LIN {X 0,Y 351.942,Z 392.186,A -85,B 0,C 180,E1 14008.468,E2 14008.468} C_VEL
LIN {X 0,Y 334.172,Z 595.574,A -85,B 0,C 180,E1 14003.413,E2 14003.413} C_VEL
LIN {X 0,Y 330.821,Z 619.274,A -85,B 0,C 180,E1 14002.569,E2 14002.569} C_VEL
LIN {X 0,Y 326.72,Z 641.204,A -85,B 0,C 180,E1 14001.516,E2 14001.516} C_VEL
LIN {X 0,Y 321.807,Z 663.482,A -85,B 0,C 180,E1 14000.12,E2 14000.12} C_VEL
LIN {X 0,Y 316.522,Z 684.324,A -85,B 0,C 180,E1 13998.471,E2 13998.471} C_VEL
LIN {X 0,Y 310.9,Z 704.371,A -85,B 0,C 180,E1 13996.508,E2 13996.508} C_VEL
LIN {X 0,Y 304.922,Z 723.772,A -85,B 0,C 180,E1 13994.168,E2 13994.168} C_VEL
LIN {X 0,Y 299.118,Z 741.54,A -85,B 0,C 180,E1 13991.566,E2 13991.566} C_VEL
LIN {X 0,Y 293.223,Z 758.965,A -85,B 0,C 180,E1 13988.482,E2 13988.482} C_VEL
LIN {X 0,Y 288.236,Z 773.54,A -85,B 0,C 180,E1 13985.391,E2 13985.391} C_VEL
LIN {X 0,Y 283.487,Z 787.604,A -85,B 0,C 180,E1 13981.785,E2 13981.785} C_VEL
LIN {X 0,Y 279.718,Z 799.334,A -85,B 0,C 180,E1 13978.151,E2 13978.151} C_VEL
LIN {X 0,Y 276.584,Z 810.131,A -85,B 0,C 180,E1 13974.108,E2 13974.108} C_VEL
LIN {X 0,Y 274.424,Z 818.988,A -85,B 0,C 180,E1 13970.026,E2 13970.026} C_VEL
LIN {X 0,Y 273.126,Z 825.97,A -85,B 0,C 180,E1 13965.933,E2 13965.933} C_VEL
LIN {X 0,Y 272.509,Z 831.598,A -85,B 0,C 180,E1 13961.64,E2 13961.64} C_VEL
LIN {X 0,Y 272.417,Z 835.097,A -85,B 0,C 180,E1 13957.803,E2 13957.803} C_VEL
LIN {X 0,Y 272.52,Z 837.318,A -85,B 0,C 180,E1 13953.784,E2 13953.784} C_VEL
LIN {X 0,Y 272.599,Z 837.937,A -85,B 0,C 180,E1 13950.208,E2 13950.208} C_VEL
LIN {X 0,Y 272.53,Z 837.335,A -85,B 0,C 180,E1 13946.422,E2 13946.422} C_VEL
LIN {X 0,Y 272.421,Z 835.096,A -85,B 0,C 180,E1 13942.405,E2 13942.405} C_VEL
LIN {X 0,Y 272.503,Z 831.449,A -85,B 0,C 180,E1 13938.356,E2 13938.356} C_VEL
LIN {X 0,Y 273.106,Z 825.844,A -85,B 0,C 180,E1 13934.061,E2 13934.061} C_VEL
LIN {X 0,Y 274.571,Z 818.159,A -85,B 0,C 180,E1 13929.536,E2 13929.536} C_VEL
LIN {X 0,Y 276.978,Z 808.952,A -85,B 0,C 180,E1 13925.243,E2 13925.243} C_VEL
LIN {X 0,Y 280.51,Z 797.735,A -85,B 0,C 180,E1 13921.001,E2 13921.001} C_VEL
LIN {X 0,Y 285.267,Z 784.462,A -85,B 0,C 180,E1 13916.852,E2 13916.852} C_VEL
LIN {X 0,Y 290.991,Z 769.791,A -85,B 0,C 180,E1 13913.034,E2 13913.034} C_VEL
LIN {X 0,Y 298.348,Z 751.957,A -85,B 0,C 180,E1 13909.192,E2 13909.192} C_VEL
LIN {X 0,Y 307.129,Z 731.579,A -85,B 0,C 180,E1 13905.577,E2 13905.577} C_VEL
LIN {X 0,Y 316.878,Z 709.867,A -85,B 0,C 180,E1 13902.407,E2 13902.407} C_VEL
LIN {X 0,Y 327.837,Z 686.66,A -85,B 0,C 180,E1 13899.636,E2 13899.636} C_VEL
LIN {X 0,Y 339.629,Z 663.013,A -85,B 0,C 180,E1 13897.355,E2 13897.355} C_VEL
LIN {X 0,Y 346.995,Z 648.595,A -85,B 0,C 180,E1 13896.209,E2 13896.209} C_VEL
LIN {X 0,Y 335.989,Z 668.452,A -85,B 0,C 180,E1 13894.02,E2 13894.02} C_VEL
LIN {X 0,Y 324.563,Z 689.118,A -85,B 0,C 180,E1 13891.17,E2 13891.17} C_VEL
LIN {X 0,Y 315.027,Z 706.467,A -85,B 0,C 180,E1 13888.225,E2 13888.225} C_VEL
LIN {X 0,Y 305.764,Z 723.244,A -85,B 0,C 180,E1 13884.746,E2 13884.746} C_VEL
LIN {X 0,Y 298.466,Z 736.332,A -85,B 0,C 180,E1 13881.419,E2 13881.419} C_VEL
LIN {X 0,Y 291.857,Z 748.263,A -85,B 0,C 180,E1 13877.755,E2 13877.755} C_VEL
LIN {X 0,Y 286.081,Z 758.861,A -85,B 0,C 180,E1 13873.751,E2 13873.751} C_VEL
LIN {X 0,Y 281.081,Z 768.361,A -85,B 0,C 180,E1 13869.214,E2 13869.214} C_VEL
LIN {X 0,Y 277.403,Z 775.806,A -85,B 0,C 180,E1 13864.551,E2 13864.551} C_VEL
LIN {X 0,Y 275.095,Z 780.905,A -85,B 0,C 180,E1 13860.211,E2 13860.211} C_VEL
LIN {X 0,Y 273.648,Z 784.687,A -85,B 0,C 180,E1 13855.602,E2 13855.602} C_VEL
LIN {X 0,Y 272.931,Z 786.813,A -85,B 0,C 180,E1 13851.152,E2 13851.152} C_VEL
LIN {X 0,Y 272.65,Z 787.32,A -85,B 0,C 180,E1 13847.077,E2 13847.077} C_VEL
LIN {X 0,Y 272.588,Z 786.619,A -85,B 0,C 180,E1 13842.939,E2 13842.939} C_VEL
LIN {X 0,Y 272.677,Z 784.598,A -85,B 0,C 180,E1 13838.943,E2 13838.943} C_VEL
LIN {X 0,Y 273.155,Z 780.795,A -85,B 0,C 180,E1 13834.414,E2 13834.414} C_VEL
LIN {X 0,Y 274.12,Z 775.808,A -85,B 0,C 180,E1 13830.243,E2 13830.243} C_VEL
LIN {X 0,Y 275.777,Z 769.08,A -85,B 0,C 180,E1 13826.063,E2 13826.063} C_VEL
LIN {X 0,Y 278.331,Z 760.51,A -85,B 0,C 180,E1 13821.843,E2 13821.843} C_VEL
LIN {X 0,Y 281.677,Z 750.53,A -85,B 0,C 180,E1 13817.87,E2 13817.87} C_VEL
LIN {X 0,Y 285.732,Z 739.008,A -85,B 0,C 180,E1 13814.138,E2 13814.138} C_VEL
LIN {X 0,Y 290.521,Z 725.684,A -85,B 0,C 180,E1 13810.578,E2 13810.578} C_VEL
LIN {X 0,Y 296.06,Z 710.191,A -85,B 0,C 180,E1 13807.159,E2 13807.159} C_VEL
LIN {X 0,Y 301.439,Z 694.762,A -85,B 0,C 180,E1 13804.325,E2 13804.325} C_VEL
LIN {X 0,Y 307.215,Z 677.128,A -85,B 0,C 180,E1 13801.637,E2 13801.637} C_VEL
LIN {X 0,Y 312.723,Z 658.939,A -85,B 0,C 180,E1 13799.343,E2 13799.343} C_VEL
LIN {X 0,Y 318.43,Z 638.248,A -85,B 0,C 180,E1 13797.194,E2 13797.194} C_VEL
LIN {X 0,Y 323.465,Z 617.601,A -85,B 0,C 180,E1 13795.448,E2 13795.448} C_VEL
LIN {X 0,Y 327.941,Z 596.27,A -85,B 0,C 180,E1 13793.992,E2 13793.992} C_VEL
LIN {X 0,Y 331.872,Z 573.214,A -85,B 0,C 180,E1 13792.774,E2 13792.774} C_VEL
LIN {X 0,Y 334.859,Z 550.767,A -85,B 0,C 180,E1 13791.893,E2 13791.893} C_VEL
LIN {X 0,Y 337.662,Z 520.747,A -85,B 0,C 180,E1 13791.075,E2 13791.075} C_VEL
LIN {X 0,Y 349.694,Z 379.97,A -85,B 0,C 180,E1 13787.623,E2 13787.623} C_VEL
LIN {X 0,Y 338.542,Z 362.97,A -85,B 0,C 180,E1 13784.541,E2 13784.541} C_VEL
LIN {X 0,Y 328.746,Z 348.783,A -85,B 0,C 180,E1 13781.553,E2 13781.553} C_VEL
LIN {X 0,Y 319.208,Z 335.537,A -85,B 0,C 180,E1 13778.335,E2 13778.335} C_VEL
LIN {X 0,Y 311.113,Z 324.801,A -85,B 0,C 180,E1 13775.303,E2 13775.303} C_VEL
LIN {X 0,Y 307.024,Z 319.574,A -85,B 0,C 180,E1 13773.69,E2 13773.69} C_VEL
LIN {X 0,Y 303.123,Z 314.492,A -85,B 0,C 180,E1 13772.013,E2 13772.013} C_VEL
LIN {X 0,Y 298.721,Z 308.948,A -85,B 0,C 180,E1 13770.055,E2 13770.055} C_VEL
LIN {X 0,Y 295.301,Z 304.475,A -85,B 0,C 180,E1 13768.401,E2 13768.401} C_VEL
LIN {X 0,Y 290.911,Z 299.407,A -85,B 0,C 180,E1 13766.208,E2 13766.208} C_VEL
LIN {X 0,Y 289.799,Z 297.619,A -85,B 0,C 180,E1 13765.583,E2 13765.583} C_VEL
LIN {X 0,Y 286.586,Z 294.45,A -85,B 0,C 180,E1 13763.855,E2 13763.855} C_VEL
LIN {X 0,Y 284.817,Z 291.431,A -85,B 0,C 180,E1 13762.742,E2 13762.742} C_VEL
LIN {X 0,Y 281.599,Z 288.767,A -85,B 0,C 180,E1 13760.911,E2 13760.911} C_VEL
LIN {X 0,Y 279.649,Z 285.071,A -85,B 0,C 180,E1 13759.472,E2 13759.472} C_VEL
LIN {X 0,Y 276.423,Z 282.89,A -85,B 0,C 180,E1 13757.468,E2 13757.468} C_VEL
LIN {X 0,Y 274.693,Z 279.757,A -85,B 0,C 180,E1 13756.048,E2 13756.048} C_VEL
LIN {X 0,Y 274.436,Z 278.542,A -85,B 0,C 180,E1 13755.658,E2 13755.658} C_VEL
LIN {X 0,Y 274.453,Z 278.534,A -85,B 0,C 180,E1 13750.862,E2 13750.862} C_VEL
LIN {X 0,Y 274.454,Z 278.532,A -85,B 0,C 180,E1 13746.15,E2 13746.15} C_VEL
LIN {X 0,Y 274.433,Z 278.536,A -85,B 0,C 180,E1 13741.4,E2 13741.4} C_VEL
LIN {X 0,Y 274.449,Z 278.537,A -85,B 0,C 180,E1 13736.628,E2 13736.628} C_VEL
LIN {X 0,Y 274.445,Z 278.542,A -85,B 0,C 180,E1 13731.893,E2 13731.893} C_VEL
LIN {X 0,Y 274.427,Z 278.549,A -85,B 0,C 180,E1 13727.077,E2 13727.077} C_VEL
LIN {X 0,Y 274.45,Z 278.55,A -85,B 0,C 180,E1 13722.31,E2 13722.31} C_VEL
LIN {X 0,Y 274.443,Z 278.549,A -85,B 0,C 180,E1 13717.734,E2 13717.734} C_VEL
LIN {X 0,Y 274.423,Z 278.554,A -85,B 0,C 180,E1 13712.876,E2 13712.876} C_VEL
LIN {X 0,Y 274.445,Z 278.55,A -85,B 0,C 180,E1 13708.163,E2 13708.163} C_VEL
LIN {X 0,Y 274.429,Z 278.552,A -85,B 0,C 180,E1 13703.351,E2 13703.351} C_VEL
LIN {X 0,Y 274.442,Z 278.55,A -85,B 0,C 180,E1 13699.818,E2 13699.818} C_VEL
LIN {X 0,Y 273.594,Z 278.663,A -85,B 0,C 180,E1 13698.323,E2 13698.323} C_VEL
LIN {X 0,Y 269.921,Z 279.115,A -85,B 0,C 180,E1 13695.846,E2 13695.846} C_VEL
LIN {X 0,Y 266.816,Z 279.496,A -85,B 0,C 180,E1 13693.407,E2 13693.407} C_VEL
LIN {X 0,Y 266.475,Z 279.543,A -85,B 0,C 180,E1 13692.444,E2 13692.444} C_VEL
LIN {X 0,Y 266.523,Z 279.674,A -85,B 0,C 180,E1 13687.704,E2 13687.704} C_VEL
LIN {X 0,Y 267.429,Z 282.454,A -85,B 0,C 180,E1 13686.545,E2 13686.545} C_VEL
LIN {X 0,Y 270.123,Z 285.3,A -85,B 0,C 180,E1 13684.243,E2 13684.243} C_VEL
LIN {X 0,Y 272.079,Z 286.502,A -85,B 0,C 180,E1 13682.788,E2 13682.788} C_VEL
LIN {X 0,Y 274,Z 290.15,A -85,B 0,C 180,E1 13681.121,E2 13681.121} C_VEL
LIN {X 0,Y 277.469,Z 293.008,A -85,B 0,C 180,E1 13678.758,E2 13678.758} C_VEL
LIN {X 0,Y 279.723,Z 296.759,A -85,B 0,C 180,E1 13677.129,E2 13677.129} C_VEL
LIN {X 0,Y 282.798,Z 299.497,A -85,B 0,C 180,E1 13675.282,E2 13675.282} C_VEL
LIN {X 0,Y 285.389,Z 303.379,A -85,B 0,C 180,E1 13673.661,E2 13673.661} C_VEL
LIN {X 0,Y 287.285,Z 305.462,A -85,B 0,C 180,E1 13672.599,E2 13672.599} C_VEL
LIN {X 0,Y 291.204,Z 310.688,A -85,B 0,C 180,E1 13670.412,E2 13670.412} C_VEL
LIN {X 0,Y 295.841,Z 316.996,A -85,B 0,C 180,E1 13668.051,E2 13668.051} C_VEL
LIN {X 0,Y 302.81,Z 326.638,A -85,B 0,C 180,E1 13664.779,E2 13664.779} C_VEL
LIN {X 0,Y 312.198,Z 340.01,A -85,B 0,C 180,E1 13660.834,E2 13660.834} C_VEL
LIN {X 0,Y 322.538,Z 355.803,A -85,B 0,C 180,E1 13656.958,E2 13656.958} C_VEL
LIN {X 0,Y 332.5,Z 371.552,A -85,B 0,C 180,E1 13653.62,E2 13653.62} C_VEL
LIN {X 0,Y 343.151,Z 389.583,A -85,B 0,C 180,E1 13650.378,E2 13650.378} C_VEL
LIN {X 0,Y 346.545,Z 395.753,A -85,B 0,C 180,E1 13649.4,E2 13649.4} C_VEL
LIN {X 0,Y 328.463,Z 594.891,A -85,B 0,C 180,E1 13644.391,E2 13644.391} C_VEL
LIN {X 0,Y 324.989,Z 618.714,A -85,B 0,C 180,E1 13643.533,E2 13643.533} C_VEL
LIN {X 0,Y 320.71,Z 640.907,A -85,B 0,C 180,E1 13642.457,E2 13642.457} C_VEL
LIN {X 0,Y 315.639,Z 663.183,A -85,B 0,C 180,E1 13641.045,E2 13641.045} C_VEL
LIN {X 0,Y 310.162,Z 684.106,A -85,B 0,C 180,E1 13639.367,E2 13639.367} C_VEL
LIN {X 0,Y 304.352,Z 704.148,A -85,B 0,C 180,E1 13637.379,E2 13637.379} C_VEL
LIN {X 0,Y 298.224,Z 723.376,A -85,B 0,C 180,E1 13635.022,E2 13635.022} C_VEL
LIN {X 0,Y 292.219,Z 741.11,A -85,B 0,C 180,E1 13632.378,E2 13632.378} C_VEL
LIN {X 0,Y 286.097,Z 758.503,A -85,B 0,C 180,E1 13629.236,E2 13629.236} C_VEL
LIN {X 0,Y 280.773,Z 773.445,A -85,B 0,C 180,E1 13625.982,E2 13625.982} C_VEL
LIN {X 0,Y 276.01,Z 787.001,A -85,B 0,C 180,E1 13622.418,E2 13622.418} C_VEL
LIN {X 0,Y 271.94,Z 799.128,A -85,B 0,C 180,E1 13618.551,E2 13618.551} C_VEL
LIN {X 0,Y 268.556,Z 810.359,A -85,B 0,C 180,E1 13614.173,E2 13614.173} C_VEL
LIN {X 0,Y 266.376,Z 819.075,A -85,B 0,C 180,E1 13609.97,E2 13609.97} C_VEL
LIN {X 0,Y 265.086,Z 825.898,A -85,B 0,C 180,E1 13605.755,E2 13605.755} C_VEL
LIN {X 0,Y 264.51,Z 831.309,A -85,B 0,C 180,E1 13601.334,E2 13601.334} C_VEL
LIN {X 0,Y 264.453,Z 834.685,A -85,B 0,C 180,E1 13597.383,E2 13597.383} C_VEL
LIN {X 0,Y 264.572,Z 836.606,A -85,B 0,C 180,E1 13593.464,E2 13593.464} C_VEL
LIN {X 0,Y 264.645,Z 837.141,A -85,B 0,C 180,E1 13589.998,E2 13589.998} C_VEL
LIN {X 0,Y 264.552,Z 836.49,A -85,B 0,C 180,E1 13586.097,E2 13586.097} C_VEL
LIN {X 0,Y 264.439,Z 834.34,A -85,B 0,C 180,E1 13582.164,E2 13582.164} C_VEL
LIN {X 0,Y 264.522,Z 830.928,A -85,B 0,C 180,E1 13578.22,E2 13578.22} C_VEL
LIN {X 0,Y 265.211,Z 825.167,A -85,B 0,C 180,E1 13573.573,E2 13573.573} C_VEL
LIN {X 0,Y 266.716,Z 817.962,A -85,B 0,C 180,E1 13569.135,E2 13569.135} C_VEL
LIN {X 0,Y 269.273,Z 808.87,A -85,B 0,C 180,E1 13564.72,E2 13564.72} C_VEL
LIN {X 0,Y 273.259,Z 797.259,A -85,B 0,C 180,E1 13560.136,E2 13560.136} C_VEL
LIN {X 0,Y 278.636,Z 783.539,A -85,B 0,C 180,E1 13555.708,E2 13555.708} C_VEL
LIN {X 0,Y 285.158,Z 768.226,A -85,B 0,C 180,E1 13551.637,E2 13551.637} C_VEL
LIN {X 0,Y 293.535,Z 749.713,A -85,B 0,C 180,E1 13547.587,E2 13547.587} C_VEL
LIN {X 0,Y 303.996,Z 727.824,A -85,B 0,C 180,E1 13543.688,E2 13543.688} C_VEL
LIN {X 0,Y 315.653,Z 704.899,A -85,B 0,C 180,E1 13540.375,E2 13540.375} C_VEL
LIN {X 0,Y 327.969,Z 682.1,A -85,B 0,C 180,E1 13537.708,E2 13537.708} C_VEL
LIN {X 0,Y 337.842,Z 664.742,A -85,B 0,C 180,E1 13536.037,E2 13536.037} C_VEL
LIN {X 0,Y 325.213,Z 684.979,A -85,B 0,C 180,E1 13533.392,E2 13533.392} C_VEL
LIN {X 0,Y 313.431,Z 704.056,A -85,B 0,C 180,E1 13530.269,E2 13530.269} C_VEL
LIN {X 0,Y 302.725,Z 721.589,A -85,B 0,C 180,E1 13526.694,E2 13526.694} C_VEL
LIN {X 0,Y 293.873,Z 736.129,A -85,B 0,C 180,E1 13523.036,E2 13523.036} C_VEL
LIN {X 0,Y 286.647,Z 748.093,A -85,B 0,C 180,E1 13519.354,E2 13519.354} C_VEL
LIN {X 0,Y 279.981,Z 759.214,A -85,B 0,C 180,E1 13515.114,E2 13515.114} C_VEL
LIN {X 0,Y 274.435,Z 768.713,A -85,B 0,C 180,E1 13510.499,E2 13510.499} C_VEL
LIN {X 0,Y 270.449,Z 775.926,A -85,B 0,C 180,E1 13505.944,E2 13505.944} C_VEL
LIN {X 0,Y 267.672,Z 781.44,A -85,B 0,C 180,E1 13501.287,E2 13501.287} C_VEL
LIN {X 0,Y 266.015,Z 785.203,A -85,B 0,C 180,E1 13496.771,E2 13496.771} C_VEL
LIN {X 0,Y 265.136,Z 787.339,A -85,B 0,C 180,E1 13492.419,E2 13492.419} C_VEL
LIN {X 0,Y 264.721,Z 788.143,A -85,B 0,C 180,E1 13487.792,E2 13487.792} C_VEL
LIN {X 0,Y 264.624,Z 787.62,A -85,B 0,C 180,E1 13483.767,E2 13483.767} C_VEL
LIN {X 0,Y 264.686,Z 785.665,A -85,B 0,C 180,E1 13479.436,E2 13479.436} C_VEL
LIN {X 0,Y 265.091,Z 782.273,A -85,B 0,C 180,E1 13475.015,E2 13475.015} C_VEL
LIN {X 0,Y 266.004,Z 777.39,A -85,B 0,C 180,E1 13470.7,E2 13470.7} C_VEL
LIN {X 0,Y 267.726,Z 770.585,A -85,B 0,C 180,E1 13466.193,E2 13466.193} C_VEL
LIN {X 0,Y 270.302,Z 762.203,A -85,B 0,C 180,E1 13461.853,E2 13461.853} C_VEL
LIN {X 0,Y 273.697,Z 752.363,A -85,B 0,C 180,E1 13457.769,E2 13457.769} C_VEL
LIN {X 0,Y 277.793,Z 741.088,A -85,B 0,C 180,E1 13453.963,E2 13453.963} C_VEL
LIN {X 0,Y 282.93,Z 727.351,A -85,B 0,C 180,E1 13450.142,E2 13450.142} C_VEL
LIN {X 0,Y 288.379,Z 712.726,A -85,B 0,C 180,E1 13446.789,E2 13446.789} C_VEL
LIN {X 0,Y 294.323,Z 696.294,A -85,B 0,C 180,E1 13443.671,E2 13443.671} C_VEL
LIN {X 0,Y 300.189,Z 678.978,A -85,B 0,C 180,E1 13440.97,E2 13440.97} C_VEL
LIN {X 0,Y 305.923,Z 660.788,A -85,B 0,C 180,E1 13438.611,E2 13438.611} C_VEL
LIN {X 0,Y 311.642,Z 640.918,A -85,B 0,C 180,E1 13436.483,E2 13436.483} C_VEL
LIN {X 0,Y 316.902,Z 620.387,A -85,B 0,C 180,E1 13434.687,E2 13434.687} C_VEL
LIN {X 0,Y 321.588,Z 598.842,A -85,B 0,C 180,E1 13433.181,E2 13433.181} C_VEL
LIN {X 0,Y 325.565,Z 576.701,A -85,B 0,C 180,E1 13431.964,E2 13431.964} C_VEL
LIN {X 0,Y 328.935,Z 553.047,A -85,B 0,C 180,E1 13430.989,E2 13430.989} C_VEL
LIN {X 0,Y 331.69,Z 525.923,A -85,B 0,C 180,E1 13430.213,E2 13430.213} C_VEL
LIN {X 0,Y 344.309,Z 383.812,A -85,B 0,C 180,E1 13426.688,E2 13426.688} C_VEL
LIN {X 0,Y 332.876,Z 366.29,A -85,B 0,C 180,E1 13423.4,E2 13423.4} C_VEL
LIN {X 0,Y 322.598,Z 351.536,A -85,B 0,C 180,E1 13420.132,E2 13420.132} C_VEL
LIN {X 0,Y 312.829,Z 337.953,A -85,B 0,C 180,E1 13416.66,E2 13416.66} C_VEL
LIN {X 0,Y 304.199,Z 326.687,A -85,B 0,C 180,E1 13413.252,E2 13413.252} C_VEL
LIN {X 0,Y 300.032,Z 321.302,A -85,B 0,C 180,E1 13411.442,E2 13411.442} C_VEL
LIN {X 0,Y 295.841,Z 315.95,A -85,B 0,C 180,E1 13409.527,E2 13409.527} C_VEL
LIN {X 0,Y 291.65,Z 310.532,A -85,B 0,C 180,E1 13407.448,E2 13407.448} C_VEL
LIN {X 0,Y 288.18,Z 306.433,A -85,B 0,C 180,E1 13405.674,E2 13405.674} C_VEL
LIN {X 0,Y 286.993,Z 304.767,A -85,B 0,C 180,E1 13405.005,E2 13405.005} C_VEL
LIN {X 0,Y 283.721,Z 301.163,A -85,B 0,C 180,E1 13403.176,E2 13403.176} C_VEL
LIN {X 0,Y 282.258,Z 298.807,A -85,B 0,C 180,E1 13402.266,E2 13402.266} C_VEL
LIN {X 0,Y 279.069,Z 295.873,A -85,B 0,C 180,E1 13400.36,E2 13400.36} C_VEL
LIN {X 0,Y 277.159,Z 292.56,A -85,B 0,C 180,E1 13398.979,E2 13398.979} C_VEL
LIN {X 0,Y 273.841,Z 289.901,A -85,B 0,C 180,E1 13396.811,E2 13396.811} C_VEL
LIN {X 0,Y 271.834,Z 286.096,A -85,B 0,C 180,E1 13395.082,E2 13395.082} C_VEL
LIN {X 0,Y 268.572,Z 283.959,A -85,B 0,C 180,E1 13392.675,E2 13392.675} C_VEL
LIN {X 0,Y 266.903,Z 281.204,A -85,B 0,C 180,E1 13391.038,E2 13391.038} C_VEL
LIN {X 0,Y 266.52,Z 279.52,A -85,B 0,C 180,E1 13390.498,E2 13390.498} C_VEL
LIN {X 0,Y 266.498,Z 279.523,A -85,B 0,C 180,E1 13385.731,E2 13385.731} C_VEL
LIN {X 0,Y 266.508,Z 279.527,A -85,B 0,C 180,E1 13380.812,E2 13380.812} C_VEL
LIN {X 0,Y 266.507,Z 279.533,A -85,B 0,C 180,E1 13376.002,E2 13376.002} C_VEL
LIN {X 0,Y 266.489,Z 279.542,A -85,B 0,C 180,E1 13371.205,E2 13371.205} C_VEL
LIN {X 0,Y 266.51,Z 279.544,A -85,B 0,C 180,E1 13366.349,E2 13366.349} C_VEL
LIN {X 0,Y 266.495,Z 279.547,A -85,B 0,C 180,E1 13361.607,E2 13361.607} C_VEL
LIN {X 0,Y 266.492,Z 279.542,A -85,B 0,C 180,E1 13356.596,E2 13356.596} C_VEL
LIN {X 0,Y 266.509,Z 279.537,A -85,B 0,C 180,E1 13351.933,E2 13351.933} C_VEL
LIN {X 0,Y 266.486,Z 279.536,A -85,B 0,C 180,E1 13347.23,E2 13347.23} C_VEL
LIN {X 0,Y 266.492,Z 279.531,A -85,B 0,C 180,E1 13342.265,E2 13342.265} C_VEL
LIN {X 0,Y 266.492,Z 279.528,A -85,B 0,C 180,E1 13337.463,E2 13337.463} C_VEL
LIN {X 0,Y 266.474,Z 279.543,A -85,B 0,C 180,E1 13332.566,E2 13332.566} C_VEL
LIN {X 0,Y 266.475,Z 279.543,A -85,B 0,C 180,E1 13332.444,E2 13332.444} C_VEL
LIN {X 0,Y 266.106,Z 280.303,A -85,B 0,C 180,E1 13331.338,E2 13331.338} C_VEL
LIN {X 0,Y 264.864,Z 283.505,A -85,B 0,C 180,E1 13329.703,E2 13329.703} C_VEL
LIN {X 0,Y 264.474,Z 287.92,A -85,B 0,C 180,E1 13327.957,E2 13327.957} C_VEL
LIN {X 0,Y 264.679,Z 288.591,A -85,B 0,C 180,E1 13327.663,E2 13327.663} C_VEL
LIN {X 0,Y 266.748,Z 291.851,A -85,B 0,C 180,E1 13325.59,E2 13325.59} C_VEL
LIN {X 0,Y 269.783,Z 294.028,A -85,B 0,C 180,E1 13323.237,E2 13323.237} C_VEL
LIN {X 0,Y 272.021,Z 297.888,A -85,B 0,C 180,E1 13321.333,E2 13321.333} C_VEL
LIN {X 0,Y 275.163,Z 300.601,A -85,B 0,C 180,E1 13319.164,E2 13319.164} C_VEL
LIN {X 0,Y 277.712,Z 304.517,A -85,B 0,C 180,E1 13317.315,E2 13317.315} C_VEL
LIN {X 0,Y 280.388,Z 306.967,A -85,B 0,C 180,E1 13315.703,E2 13315.703} C_VEL
LIN {X 0,Y 283.392,Z 311.177,A -85,B 0,C 180,E1 13313.82,E2 13313.82} C_VEL
LIN {X 0,Y 285.203,Z 313.416,A -85,B 0,C 180,E1 13312.787,E2 13312.787} C_VEL
LIN {X 0,Y 288.592,Z 317.897,A -85,B 0,C 180,E1 13310.883,E2 13310.883} C_VEL
LIN {X 0,Y 293.267,Z 324.376,A -85,B 0,C 180,E1 13308.443,E2 13308.443} C_VEL
LIN {X 0,Y 299.789,Z 333.498,A -85,B 0,C 180,E1 13305.314,E2 13305.314} C_VEL
LIN {X 0,Y 308.896,Z 346.614,A -85,B 0,C 180,E1 13301.405,E2 13301.405} C_VEL
LIN {X 0,Y 318.934,Z 362.103,A -85,B 0,C 180,E1 13297.56,E2 13297.56} C_VEL
LIN {X 0,Y 328.594,Z 377.505,A -85,B 0,C 180,E1 13294.253,E2 13294.253} C_VEL
LIN {X 0,Y 339.211,Z 395.689,A -85,B 0,C 180,E1 13290.945,E2 13290.945} C_VEL
LIN {X 0,Y 341.176,Z 399.501,A -85,B 0,C 180,E1 13290.351,E2 13290.351} C_VEL
LIN {X 0,Y 322.724,Z 594.496,A -85,B 0,C 180,E1 13285.377,E2 13285.377} C_VEL
LIN {X 0,Y 319.149,Z 618.283,A -85,B 0,C 180,E1 13284.511,E2 13284.511} C_VEL
LIN {X 0,Y 314.705,Z 640.646,A -85,B 0,C 180,E1 13283.415,E2 13283.415} C_VEL
LIN {X 0,Y 309.548,Z 662.612,A -85,B 0,C 180,E1 13282.008,E2 13282.008} C_VEL
LIN {X 0,Y 303.765,Z 684.004,A -85,B 0,C 180,E1 13280.269,E2 13280.269} C_VEL
LIN {X 0,Y 297.664,Z 704.298,A -85,B 0,C 180,E1 13278.216,E2 13278.216} C_VEL
LIN {X 0,Y 291.356,Z 723.49,A -85,B 0,C 180,E1 13275.823,E2 13275.823} C_VEL
LIN {X 0,Y 285.164,Z 741.146,A -85,B 0,C 180,E1 13273.132,E2 13273.132} C_VEL
LIN {X 0,Y 279.019,Z 757.975,A -85,B 0,C 180,E1 13270.03,E2 13270.03} C_VEL
LIN {X 0,Y 273.654,Z 772.52,A -85,B 0,C 180,E1 13266.81,E2 13266.81} C_VEL
LIN {X 0,Y 268.603,Z 786.3,A -85,B 0,C 180,E1 13263.115,E2 13263.115} C_VEL
LIN {X 0,Y 264.381,Z 798.3,A -85,B 0,C 180,E1 13259.197,E2 13259.197} C_VEL
LIN {X 0,Y 260.964,Z 809.063,A -85,B 0,C 180,E1 13254.924,E2 13254.924} C_VEL
LIN {X 0,Y 258.605,Z 817.905,A -85,B 0,C 180,E1 13250.597,E2 13250.597} C_VEL
LIN {X 0,Y 257.196,Z 824.874,A -85,B 0,C 180,E1 13246.209,E2 13246.209} C_VEL
LIN {X 0,Y 256.557,Z 830.34,A -85,B 0,C 180,E1 13241.69,E2 13241.69} C_VEL
LIN {X 0,Y 256.484,Z 833.764,A -85,B 0,C 180,E1 13237.614,E2 13237.614} C_VEL
LIN {X 0,Y 256.607,Z 835.774,A -85,B 0,C 180,E1 13233.572,E2 13233.572} C_VEL
LIN {X 0,Y 256.686,Z 836.331,A -85,B 0,C 180,E1 13229.998,E2 13229.998} C_VEL
LIN {X 0,Y 256.591,Z 835.761,A -85,B 0,C 180,E1 13226.2,E2 13226.2} C_VEL
LIN {X 0,Y 256.454,Z 833.617,A -85,B 0,C 180,E1 13221.929,E2 13221.929} C_VEL
LIN {X 0,Y 256.556,Z 830.211,A -85,B 0,C 180,E1 13217.849,E2 13217.849} C_VEL
LIN {X 0,Y 257.324,Z 824.493,A -85,B 0,C 180,E1 13213.055,E2 13213.055} C_VEL
LIN {X 0,Y 258.988,Z 817.376,A -85,B 0,C 180,E1 13208.482,E2 13208.482} C_VEL
LIN {X 0,Y 261.763,Z 808.355,A -85,B 0,C 180,E1 13203.941,E2 13203.941} C_VEL
LIN {X 0,Y 266.045,Z 796.958,A -85,B 0,C 180,E1 13199.26,E2 13199.26} C_VEL
LIN {X 0,Y 271.52,Z 784.19,A -85,B 0,C 180,E1 13194.936,E2 13194.936} C_VEL
LIN {X 0,Y 278.383,Z 769.264,A -85,B 0,C 180,E1 13190.79,E2 13190.79} C_VEL
LIN {X 0,Y 287.176,Z 751.446,A -85,B 0,C 180,E1 13186.692,E2 13186.692} C_VEL
LIN {X 0,Y 297.926,Z 730.952,A -85,B 0,C 180,E1 13182.834,E2 13182.834} C_VEL
LIN {X 0,Y 310.558,Z 708.587,A -85,B 0,C 180,E1 13179.402,E2 13179.402} C_VEL
LIN {X 0,Y 323.711,Z 686.923,A -85,B 0,C 180,E1 13176.722,E2 13176.722} C_VEL
LIN {X 0,Y 328.633,Z 679.199,A -85,B 0,C 180,E1 13175.863,E2 13175.863} C_VEL
LIN {X 0,Y 314.914,Z 698.765,A -85,B 0,C 180,E1 13172.885,E2 13172.885} C_VEL
LIN {X 0,Y 302.762,Z 716.583,A -85,B 0,C 180,E1 13169.479,E2 13169.479} C_VEL
LIN {X 0,Y 292.236,Z 732.229,A -85,B 0,C 180,E1 13165.757,E2 13165.757} C_VEL
LIN {X 0,Y 283.193,Z 745.764,A -85,B 0,C 180,E1 13161.762,E2 13161.762} C_VEL
LIN {X 0,Y 275.284,Z 757.737,A -85,B 0,C 180,E1 13157.33,E2 13157.33} C_VEL
LIN {X 0,Y 269.153,Z 767.239,A -85,B 0,C 180,E1 13152.881,E2 13152.881} C_VEL
LIN {X 0,Y 264.403,Z 774.959,A -85,B 0,C 180,E1 13148.265,E2 13148.265} C_VEL
LIN {X 0,Y 260.831,Z 781.171,A -85,B 0,C 180,E1 13143.299,E2 13143.299} C_VEL
LIN {X 0,Y 258.611,Z 785.354,A -85,B 0,C 180,E1 13138.452,E2 13138.452} C_VEL
LIN {X 0,Y 257.406,Z 787.89,A -85,B 0,C 180,E1 13133.759,E2 13133.759} C_VEL
LIN {X 0,Y 256.858,Z 788.991,A -85,B 0,C 180,E1 13129.234,E2 13129.234} C_VEL
LIN {X 0,Y 256.672,Z 788.625,A -85,B 0,C 180,E1 13124.874,E2 13124.874} C_VEL
LIN {X 0,Y 256.689,Z 787.009,A -85,B 0,C 180,E1 13120.432,E2 13120.432} C_VEL
LIN {X 0,Y 256.979,Z 784.029,A -85,B 0,C 180,E1 13116.116,E2 13116.116} C_VEL
LIN {X 0,Y 257.809,Z 779.365,A -85,B 0,C 180,E1 13111.513,E2 13111.513} C_VEL
LIN {X 0,Y 259.338,Z 773.318,A -85,B 0,C 180,E1 13107.074,E2 13107.074} C_VEL
LIN {X 0,Y 261.762,Z 765.344,A -85,B 0,C 180,E1 13102.608,E2 13102.608} C_VEL
LIN {X 0,Y 265.107,Z 755.766,A -85,B 0,C 180,E1 13098.313,E2 13098.313} C_VEL
LIN {X 0,Y 269.31,Z 744.602,A -85,B 0,C 180,E1 13094.236,E2 13094.236} C_VEL
LIN {X 0,Y 274.328,Z 731.727,A -85,B 0,C 180,E1 13090.387,E2 13090.387} C_VEL
LIN {X 0,Y 279.898,Z 717.262,A -85,B 0,C 180,E1 13086.859,E2 13086.859} C_VEL
LIN {X 0,Y 285.852,Z 701.374,A -85,B 0,C 180,E1 13083.652,E2 13083.652} C_VEL
LIN {X 0,Y 292.049,Z 684.074,A -85,B 0,C 180,E1 13080.767,E2 13080.767} C_VEL
LIN {X 0,Y 298.102,Z 665.944,A -85,B 0,C 180,E1 13078.262,E2 13078.262} C_VEL
LIN {X 0,Y 304.016,Z 646.359,A -85,B 0,C 180,E1 13076.044,E2 13076.044} C_VEL
LIN {X 0,Y 309.507,Z 625.976,A -85,B 0,C 180,E1 13074.163,E2 13074.163} C_VEL
LIN {X 0,Y 314.667,Z 603.891,A -85,B 0,C 180,E1 13072.521,E2 13072.521} C_VEL
LIN {X 0,Y 318.897,Z 582.26,A -85,B 0,C 180,E1 13071.248,E2 13071.248} C_VEL
LIN {X 0,Y 322.505,Z 559.319,A -85,B 0,C 180,E1 13070.214,E2 13070.214} C_VEL
LIN {X 0,Y 325.24,Z 535.374,A -85,B 0,C 180,E1 13069.455,E2 13069.455} C_VEL
LIN {X 0,Y 338.861,Z 387.588,A -85,B 0,C 180,E1 13065.731,E2 13065.731} C_VEL
LIN {X 0,Y 328.152,Z 371.194,A -85,B 0,C 180,E1 13062.54,E2 13062.54} C_VEL
LIN {X 0,Y 318.86,Z 357.651,A -85,B 0,C 180,E1 13059.477,E2 13059.477} C_VEL
LIN {X 0,Y 309.53,Z 344.557,A -85,B 0,C 180,E1 13056.074,E2 13056.074} C_VEL
LIN {X 0,Y 300.959,Z 333.282,A -85,B 0,C 180,E1 13052.62,E2 13052.62} C_VEL
LIN {X 0,Y 296.847,Z 327.999,A -85,B 0,C 180,E1 13050.83,E2 13050.83} C_VEL
LIN {X 0,Y 292.983,Z 322.945,A -85,B 0,C 180,E1 13048.994,E2 13048.994} C_VEL
LIN {X 0,Y 288.847,Z 317.623,A -85,B 0,C 180,E1 13046.926,E2 13046.926} C_VEL
LIN {X 0,Y 285.302,Z 313.162,A -85,B 0,C 180,E1 13045.026,E2 13045.026} C_VEL
LIN {X 0,Y 283.712,Z 311.406,A -85,B 0,C 180,E1 13044.136,E2 13044.136} C_VEL
LIN {X 0,Y 280.414,Z 307.115,A -85,B 0,C 180,E1 13042.215,E2 13042.215} C_VEL
LIN {X 0,Y 279.529,Z 306.031,A -85,B 0,C 180,E1 13041.673,E2 13041.673} C_VEL
LIN {X 0,Y 276.397,Z 302.752,A -85,B 0,C 180,E1 13039.698,E2 13039.698} C_VEL
LIN {X 0,Y 274.804,Z 300.066,A -85,B 0,C 180,E1 13038.565,E2 13038.565} C_VEL
LIN {X 0,Y 271.525,Z 297.2,A -85,B 0,C 180,E1 13036.322,E2 13036.322} C_VEL
LIN {X 0,Y 269.545,Z 293.678,A -85,B 0,C 180,E1 13034.661,E2 13034.661} C_VEL
LIN {X 0,Y 266.356,Z 291.339,A -85,B 0,C 180,E1 13032.188,E2 13032.188} C_VEL
LIN {X 0,Y 264.518,Z 288.257,A -85,B 0,C 180,E1 13030.402,E2 13030.402} C_VEL
LIN {X 0,Y 264.056,Z 287.139,A -85,B 0,C 180,E1 13029.882,E2 13029.882} C_VEL
LIN {X 0,Y 260.718,Z 285.035,A -85,B 0,C 180,E1 13026.736,E2 13026.736} C_VEL
LIN {X 0,Y 258.902,Z 281.985,A -85,B 0,C 180,E1 13024.485,E2 13024.485} C_VEL
LIN {X 0,Y 258.564,Z 280.53,A -85,B 0,C 180,E1 13023.775,E2 13023.775} C_VEL
LIN {X 0,Y 258.571,Z 280.52,A -85,B 0,C 180,E1 13018.705,E2 13018.705} C_VEL
LIN {X 0,Y 258.565,Z 280.518,A -85,B 0,C 180,E1 13013.913,E2 13013.913} C_VEL
LIN {X 0,Y 258.554,Z 280.517,A -85,B 0,C 180,E1 13008.901,E2 13008.901} C_VEL
LIN {X 0,Y 258.568,Z 280.515,A -85,B 0,C 180,E1 13004.012,E2 13004.012} C_VEL
LIN {X 0,Y 258.546,Z 280.516,A -85,B 0,C 180,E1 12999.072,E2 12999.072} C_VEL
LIN {X 0,Y 258.566,Z 280.513,A -85,B 0,C 180,E1 12994.1,E2 12994.1} C_VEL
LIN {X 0,Y 258.545,Z 280.517,A -85,B 0,C 180,E1 12989.157,E2 12989.157} C_VEL
LIN {X 0,Y 258.56,Z 280.52,A -85,B 0,C 180,E1 12984.138,E2 12984.138} C_VEL
LIN {X 0,Y 258.551,Z 280.53,A -85,B 0,C 180,E1 12979.346,E2 12979.346} C_VEL
LIN {X 0,Y 258.569,Z 280.753,A -85,B 0,C 180,E1 12974.481,E2 12974.481} C_VEL
LIN {X 0,Y 259.87,Z 284.059,A -85,B 0,C 180,E1 12972.552,E2 12972.552} C_VEL
LIN {X 0,Y 262.88,Z 286.674,A -85,B 0,C 180,E1 12969.41,E2 12969.41} C_VEL
LIN {X 0,Y 264.327,Z 287.545,A -85,B 0,C 180,E1 12968.097,E2 12968.097} C_VEL
LIN {X 0,Y 264.679,Z 288.591,A -85,B 0,C 180,E1 12967.663,E2 12967.663} C_VEL
LIN {X 0,Y 265.777,Z 292.988,A -85,B 0,C 180,E1 12966.175,E2 12966.175} C_VEL
LIN {X 0,Y 267.37,Z 301.032,A -85,B 0,C 180,E1 12963.86,E2 12963.86} C_VEL
LIN {X 0,Y 267.768,Z 302.085,A -85,B 0,C 180,E1 12963.442,E2 12963.442} C_VEL
LIN {X 0,Y 270.249,Z 305.85,A -85,B 0,C 180,E1 12961.375,E2 12961.375} C_VEL
LIN {X 0,Y 272.854,Z 308.117,A -85,B 0,C 180,E1 12959.577,E2 12959.577} C_VEL
LIN {X 0,Y 275.707,Z 312.26,A -85,B 0,C 180,E1 12957.503,E2 12957.503} C_VEL
LIN {X 0,Y 277.97,Z 314.396,A -85,B 0,C 180,E1 12956.13,E2 12956.13} C_VEL
LIN {X 0,Y 281.227,Z 318.789,A -85,B 0,C 180,E1 12954.079,E2 12954.079} C_VEL
LIN {X 0,Y 285.924,Z 324.99,A -85,B 0,C 180,E1 12951.4,E2 12951.4} C_VEL
LIN {X 0,Y 290.667,Z 331.726,A -85,B 0,C 180,E1 12948.841,E2 12948.841} C_VEL
LIN {X 0,Y 296.789,Z 340.355,A -85,B 0,C 180,E1 12945.86,E2 12945.86} C_VEL
LIN {X 0,Y 305.927,Z 353.728,A -85,B 0,C 180,E1 12941.86,E2 12941.86} C_VEL
LIN {X 0,Y 315.366,Z 368.402,A -85,B 0,C 180,E1 12938.175,E2 12938.175} C_VEL
LIN {X 0,Y 325.054,Z 384.053,A -85,B 0,C 180,E1 12934.783,E2 12934.783} C_VEL
LIN {X 0,Y 335.305,Z 401.883,A -85,B 0,C 180,E1 12931.501,E2 12931.501} C_VEL
LIN {X 0,Y 335.828,Z 403.24,A -85,B 0,C 180,E1 12931.322,E2 12931.322} C_VEL
LIN {X 0,Y 317.108,Z 593.923,A -85,B 0,C 180,E1 12926.405,E2 12926.405} C_VEL
LIN {X 0,Y 313.442,Z 617.632,A -85,B 0,C 180,E1 12925.533,E2 12925.533} C_VEL
LIN {X 0,Y 309.001,Z 639.398,A -85,B 0,C 180,E1 12924.464,E2 12924.464} C_VEL
LIN {X 0,Y 303.842,Z 660.89,A -85,B 0,C 180,E1 12923.092,E2 12923.092} C_VEL
LIN {X 0,Y 298.04,Z 681.956,A -85,B 0,C 180,E1 12921.39,E2 12921.39} C_VEL
LIN {X 0,Y 291.932,Z 701.759,A -85,B 0,C 180,E1 12919.4,E2 12919.4} C_VEL
LIN {X 0,Y 285.504,Z 720.738,A -85,B 0,C 180,E1 12917.045,E2 12917.045} C_VEL
LIN {X 0,Y 279.038,Z 738.738,A -85,B 0,C 180,E1 12914.322,E2 12914.322} C_VEL
LIN {X 0,Y 272.773,Z 755.347,A -85,B 0,C 180,E1 12911.281,E2 12911.281} C_VEL
LIN {X 0,Y 266.932,Z 770.607,A -85,B 0,C 180,E1 12907.898,E2 12907.898} C_VEL
LIN {X 0,Y 261.635,Z 784.37,A -85,B 0,C 180,E1 12904.175,E2 12904.175} C_VEL
LIN {X 0,Y 257.078,Z 796.767,A -85,B 0,C 180,E1 12900.111,E2 12900.111} C_VEL
LIN {X 0,Y 253.576,Z 807.221,A -85,B 0,C 180,E1 12895.953,E2 12895.953} C_VEL
LIN {X 0,Y 250.975,Z 816.22,A -85,B 0,C 180,E1 12891.498,E2 12891.498} C_VEL
LIN {X 0,Y 249.388,Z 823.383,A -85,B 0,C 180,E1 12887.016,E2 12887.016} C_VEL
LIN {X 0,Y 248.642,Z 828.914,A -85,B 0,C 180,E1 12882.539,E2 12882.539} C_VEL
LIN {X 0,Y 248.51,Z 832.598,A -85,B 0,C 180,E1 12878.195,E2 12878.195} C_VEL
LIN {X 0,Y 248.627,Z 834.783,A -85,B 0,C 180,E1 12874.149,E2 12874.149} C_VEL
LIN {X 0,Y 248.727,Z 835.523,A -85,B 0,C 180,E1 12869.998,E2 12869.998} C_VEL
LIN {X 0,Y 248.63,Z 835.031,A -85,B 0,C 180,E1 12866.309,E2 12866.309} C_VEL
LIN {X 0,Y 248.47,Z 833.029,A -85,B 0,C 180,E1 12861.87,E2 12861.87} C_VEL
LIN {X 0,Y 248.576,Z 829.716,A -85,B 0,C 180,E1 12857.689,E2 12857.689} C_VEL
LIN {X 0,Y 249.391,Z 824.2,A -85,B 0,C 180,E1 12852.739,E2 12852.739} C_VEL
LIN {X 0,Y 251.172,Z 817.188,A -85,B 0,C 180,E1 12848.024,E2 12848.024} C_VEL
LIN {X 0,Y 254.311,Z 807.937,A -85,B 0,C 180,E1 12843.117,E2 12843.117} C_VEL
LIN {X 0,Y 259.218,Z 796.053,A -85,B 0,C 180,E1 12838.061,E2 12838.061} C_VEL
LIN {X 0,Y 265.451,Z 782.856,A -85,B 0,C 180,E1 12833.476,E2 12833.476} C_VEL
LIN {X 0,Y 273.756,Z 766.616,A -85,B 0,C 180,E1 12828.894,E2 12828.894} C_VEL
LIN {X 0,Y 283.894,Z 748.177,A -85,B 0,C 180,E1 12824.646,E2 12824.646} C_VEL
LIN {X 0,Y 296.516,Z 726.849,A -85,B 0,C 180,E1 12820.648,E2 12820.648} C_VEL
LIN {X 0,Y 310.655,Z 704.923,A -85,B 0,C 180,E1 12817.345,E2 12817.345} C_VEL
LIN {X 0,Y 319.438,Z 692.138,A -85,B 0,C 180,E1 12815.718,E2 12815.718} C_VEL
LIN {X 0,Y 305.758,Z 709.754,A -85,B 0,C 180,E1 12812.656,E2 12812.656} C_VEL
LIN {X 0,Y 293.069,Z 726.57,A -85,B 0,C 180,E1 12808.979,E2 12808.979} C_VEL
LIN {X 0,Y 282.585,Z 740.704,A -85,B 0,C 180,E1 12805.127,E2 12805.127} C_VEL
LIN {X 0,Y 273.274,Z 753.454,A -85,B 0,C 180,E1 12800.79,E2 12800.79} C_VEL
LIN {X 0,Y 265.567,Z 764.131,A -85,B 0,C 180,E1 12796.18,E2 12796.18} C_VEL
LIN {X 0,Y 259.697,Z 772.552,A -85,B 0,C 180,E1 12791.552,E2 12791.552} C_VEL
LIN {X 0,Y 255.248,Z 779.286,A -85,B 0,C 180,E1 12786.752,E2 12786.752} C_VEL
LIN {X 0,Y 251.999,Z 784.473,A -85,B 0,C 180,E1 12781.595,E2 12781.595} C_VEL
LIN {X 0,Y 250.166,Z 787.671,A -85,B 0,C 180,E1 12776.796,E2 12776.796} C_VEL
LIN {X 0,Y 249.184,Z 789.489,A -85,B 0,C 180,E1 12771.93,E2 12771.93} C_VEL
LIN {X 0,Y 248.791,Z 789.788,A -85,B 0,C 180,E1 12767.469,E2 12767.469} C_VEL
LIN {X 0,Y 248.689,Z 788.825,A -85,B 0,C 180,E1 12762.936,E2 12762.936} C_VEL
LIN {X 0,Y 248.801,Z 786.62,A -85,B 0,C 180,E1 12758.553,E2 12758.553} C_VEL
LIN {X 0,Y 249.344,Z 782.756,A -85,B 0,C 180,E1 12753.83,E2 12753.83} C_VEL
LIN {X 0,Y 250.559,Z 777.31,A -85,B 0,C 180,E1 12749.091,E2 12749.091} C_VEL
LIN {X 0,Y 252.513,Z 770.564,A -85,B 0,C 180,E1 12744.658,E2 12744.658} C_VEL
LIN {X 0,Y 255.541,Z 761.7,A -85,B 0,C 180,E1 12740.078,E2 12740.078} C_VEL
LIN {X 0,Y 259.721,Z 750.676,A -85,B 0,C 180,E1 12735.526,E2 12735.526} C_VEL
LIN {X 0,Y 264.467,Z 738.802,A -85,B 0,C 180,E1 12731.539,E2 12731.539} C_VEL
LIN {X 0,Y 270.002,Z 725.073,A -85,B 0,C 180,E1 12727.774,E2 12727.774} C_VEL
LIN {X 0,Y 275.841,Z 710.279,A -85,B 0,C 180,E1 12724.436,E2 12724.436} C_VEL
LIN {X 0,Y 282.35,Z 693.134,A -85,B 0,C 180,E1 12721.241,E2 12721.241} C_VEL
LIN {X 0,Y 288.563,Z 675.745,A -85,B 0,C 180,E1 12718.567,E2 12718.567} C_VEL
LIN {X 0,Y 295.01,Z 656.172,A -85,B 0,C 180,E1 12716.093,E2 12716.093} C_VEL
LIN {X 0,Y 300.974,Z 635.825,A -85,B 0,C 180,E1 12714.006,E2 12714.006} C_VEL
LIN {X 0,Y 306.316,Z 615.069,A -85,B 0,C 180,E1 12712.28,E2 12712.28} C_VEL
LIN {X 0,Y 311.219,Z 592.743,A -85,B 0,C 180,E1 12710.798,E2 12710.798} C_VEL
LIN {X 0,Y 315.28,Z 570.209,A -85,B 0,C 180,E1 12709.64,E2 12709.64} C_VEL
LIN {X 0,Y 318.503,Z 547.245,A -85,B 0,C 180,E1 12708.764,E2 12708.764} C_VEL
LIN {X 0,Y 333.547,Z 391.505,A -85,B 0,C 180,E1 12704.763,E2 12704.763} C_VEL
LIN {X 0,Y 322.397,Z 374.372,A -85,B 0,C 180,E1 12701.314,E2 12701.314} C_VEL
LIN {X 0,Y 312.359,Z 359.907,A -85,B 0,C 180,E1 12697.867,E2 12697.867} C_VEL
LIN {X 0,Y 304.469,Z 348.976,A -85,B 0,C 180,E1 12694.853,E2 12694.853} C_VEL
LIN {X 0,Y 297.785,Z 339.969,A -85,B 0,C 180,E1 12692.022,E2 12692.022} C_VEL
LIN {X 0,Y 293.582,Z 334.534,A -85,B 0,C 180,E1 12690.148,E2 12690.148} C_VEL
LIN {X 0,Y 290.05,Z 329.826,A -85,B 0,C 180,E1 12688.406,E2 12688.406} C_VEL
LIN {X 0,Y 285.948,Z 324.594,A -85,B 0,C 180,E1 12686.343,E2 12686.343} C_VEL
LIN {X 0,Y 281.737,Z 319.197,A -85,B 0,C 180,E1 12683.993,E2 12683.993} C_VEL
LIN {X 0,Y 278.145,Z 314.798,A -85,B 0,C 180,E1 12681.891,E2 12681.891} C_VEL
LIN {X 0,Y 277.046,Z 313.365,A -85,B 0,C 180,E1 12681.19,E2 12681.19} C_VEL
LIN {X 0,Y 273.77,Z 309.757,A -85,B 0,C 180,E1 12679.103,E2 12679.103} C_VEL
LIN {X 0,Y 272.285,Z 307.437,A -85,B 0,C 180,E1 12678.028,E2 12678.028} C_VEL
LIN {X 0,Y 269.022,Z 304.247,A -85,B 0,C 180,E1 12675.693,E2 12675.693} C_VEL
LIN {X 0,Y 267.127,Z 301.167,A -85,B 0,C 180,E1 12674.129,E2 12674.129} C_VEL
LIN {X 0,Y 263.844,Z 298.36,A -85,B 0,C 180,E1 12671.441,E2 12671.441} C_VEL
LIN {X 0,Y 262.071,Z 295.001,A -85,B 0,C 180,E1 12669.629,E2 12669.629} C_VEL
LIN {X 0,Y 258.611,Z 292.514,A -85,B 0,C 180,E1 12666.294,E2 12666.294} C_VEL
LIN {X 0,Y 256.846,Z 289.367,A -85,B 0,C 180,E1 12663.967,E2 12663.967} C_VEL
LIN {X 0,Y 256.413,Z 288.229,A -85,B 0,C 180,E1 12663.239,E2 12663.239} C_VEL
LIN {X 0,Y 252.612,Z 285.845,A -85,B 0,C 180,E1 12658.239,E2 12658.239} C_VEL
LIN {X 0,Y 250.798,Z 282.409,A -85,B 0,C 180,E1 12654.325,E2 12654.325} C_VEL
LIN {X 0,Y 250.616,Z 281.505,A -85,B 0,C 180,E1 12653.53,E2 12653.53} C_VEL
LIN {X 0,Y 250.629,Z 281.503,A -85,B 0,C 180,E1 12648.533,E2 12648.533} C_VEL
LIN {X 0,Y 250.618,Z 281.505,A -85,B 0,C 180,E1 12643.64,E2 12643.64} C_VEL
LIN {X 0,Y 250.621,Z 281.506,A -85,B 0,C 180,E1 12638.484,E2 12638.484} C_VEL
LIN {X 0,Y 250.617,Z 281.508,A -85,B 0,C 180,E1 12633.512,E2 12633.512} C_VEL
LIN {X 0,Y 250.618,Z 281.515,A -85,B 0,C 180,E1 12628.339,E2 12628.339} C_VEL
LIN {X 0,Y 250.636,Z 281.735,A -85,B 0,C 180,E1 12624.697,E2 12624.697} C_VEL
LIN {X 0,Y 251.885,Z 284.925,A -85,B 0,C 180,E1 12621.538,E2 12621.538} C_VEL
LIN {X 0,Y 254.915,Z 287.655,A -85,B 0,C 180,E1 12616.864,E2 12616.864} C_VEL
LIN {X 0,Y 256.543,Z 288.485,A -85,B 0,C 180,E1 12614.87,E2 12614.87} C_VEL
LIN {X 0,Y 257.988,Z 291.802,A -85,B 0,C 180,E1 12612.759,E2 12612.759} C_VEL
LIN {X 0,Y 261.137,Z 294.48,A -85,B 0,C 180,E1 12609.473,E2 12609.473} C_VEL
LIN {X 0,Y 262.185,Z 295.222,A -85,B 0,C 180,E1 12608.495,E2 12608.495} C_VEL
LIN {X 0,Y 264.017,Z 298.657,A -85,B 0,C 180,E1 12606.521,E2 12606.521} C_VEL
LIN {X 0,Y 267.03,Z 301.142,A -85,B 0,C 180,E1 12604.077,E2 12604.077} C_VEL
LIN {X 0,Y 267.734,Z 302.008,A -85,B 0,C 180,E1 12603.476,E2 12603.476} C_VEL
LIN {X 0,Y 267.768,Z 302.085,A -85,B 0,C 180,E1 12603.442,E2 12603.442} C_VEL
LIN {X 0,Y 268.786,Z 305.893,A -85,B 0,C 180,E1 12602.271,E2 12602.271} C_VEL
LIN {X 0,Y 270.423,Z 314.939,A -85,B 0,C 180,E1 12600.143,E2 12600.143} C_VEL
LIN {X 0,Y 271.199,Z 316.787,A -85,B 0,C 180,E1 12599.475,E2 12599.475} C_VEL
LIN {X 0,Y 274.532,Z 320.721,A -85,B 0,C 180,E1 12597.179,E2 12597.179} C_VEL
LIN {X 0,Y 275.736,Z 322.169,A -85,B 0,C 180,E1 12596.411,E2 12596.411} C_VEL
LIN {X 0,Y 280.913,Z 329.036,A -85,B 0,C 180,E1 12593.217,E2 12593.217} C_VEL
LIN {X 0,Y 283.627,Z 332.71,A -85,B 0,C 180,E1 12591.687,E2 12591.687} C_VEL
LIN {X 0,Y 288.174,Z 339.198,A -85,B 0,C 180,E1 12589.199,E2 12589.199} C_VEL
LIN {X 0,Y 294.467,Z 348.25,A -85,B 0,C 180,E1 12586.098,E2 12586.098} C_VEL
LIN {X 0,Y 302.982,Z 360.834,A -85,B 0,C 180,E1 12582.323,E2 12582.323} C_VEL
LIN {X 0,Y 312.241,Z 375.402,A -85,B 0,C 180,E1 12578.636,E2 12578.636} C_VEL
LIN {X 0,Y 321.601,Z 390.78,A -85,B 0,C 180,E1 12575.28,E2 12575.28} C_VEL
LIN {X 0,Y 330.594,Z 406.509,A -85,B 0,C 180,E1 12572.333,E2 12572.333} C_VEL
LIN {X 0,Y 311.582,Z 592.95,A -85,B 0,C 180,E1 12567.47,E2 12567.47} C_VEL
LIN {X 0,Y 307.845,Z 616.541,A -85,B 0,C 180,E1 12566.597,E2 12566.597} C_VEL
LIN {X 0,Y 303.238,Z 638.563,A -85,B 0,C 180,E1 12565.515,E2 12565.515} C_VEL
LIN {X 0,Y 297.637,Z 661.199,A -85,B 0,C 180,E1 12564.052,E2 12564.052} C_VEL
LIN {X 0,Y 291.719,Z 681.973,A -85,B 0,C 180,E1 12562.345,E2 12562.345} C_VEL
LIN {X 0,Y 285.329,Z 702.055,A -85,B 0,C 180,E1 12560.295,E2 12560.295} C_VEL
LIN {X 0,Y 278.522,Z 721.48,A -85,B 0,C 180,E1 12557.83,E2 12557.83} C_VEL
LIN {X 0,Y 271.971,Z 739.041,A -85,B 0,C 180,E1 12555.099,E2 12555.099} C_VEL
LIN {X 0,Y 265.035,Z 756.72,A -85,B 0,C 180,E1 12551.744,E2 12551.744} C_VEL
LIN {X 0,Y 259.242,Z 771.273,A -85,B 0,C 180,E1 12548.382,E2 12548.382} C_VEL
LIN {X 0,Y 253.523,Z 785.66,A -85,B 0,C 180,E1 12544.328,E2 12544.328} C_VEL
LIN {X 0,Y 248.914,Z 797.713,A -85,B 0,C 180,E1 12540.137,E2 12540.137} C_VEL
LIN {X 0,Y 245.239,Z 808.349,A -85,B 0,C 180,E1 12535.602,E2 12535.602} C_VEL
LIN {X 0,Y 242.717,Z 817.063,A -85,B 0,C 180,E1 12530.999,E2 12530.999} C_VEL
LIN {X 0,Y 241.241,Z 823.876,A -85,B 0,C 180,E1 12526.367,E2 12526.367} C_VEL
LIN {X 0,Y 240.597,Z 829.218,A -85,B 0,C 180,E1 12521.504,E2 12521.504} C_VEL
LIN {X 0,Y 240.565,Z 832.521,A -85,B 0,C 180,E1 12517.16,E2 12517.16} C_VEL
LIN {X 0,Y 240.717,Z 834.297,A -85,B 0,C 180,E1 12512.855,E2 12512.855} C_VEL
LIN {X 0,Y 240.753,Z 834.696,A -85,B 0,C 180,E1 12509.284,E2 12509.284} C_VEL
LIN {X 0,Y 240.622,Z 834,A -85,B 0,C 180,E1 12505.231,E2 12505.231} C_VEL
LIN {X 0,Y 240.478,Z 831.675,A -85,B 0,C 180,E1 12500.666,E2 12500.666} C_VEL
LIN {X 0,Y 240.709,Z 828.151,A -85,B 0,C 180,E1 12496.302,E2 12496.302} C_VEL
LIN {X 0,Y 241.843,Z 822.319,A -85,B 0,C 180,E1 12491.185,E2 12491.185} C_VEL
LIN {X 0,Y 244.184,Z 814.709,A -85,B 0,C 180,E1 12486.083,E2 12486.083} C_VEL
LIN {X 0,Y 247.97,Z 805.111,A -85,B 0,C 180,E1 12481.047,E2 12481.047} C_VEL
LIN {X 0,Y 253.311,Z 793.647,A -85,B 0,C 180,E1 12476.18,E2 12476.18} C_VEL
LIN {X 0,Y 260.323,Z 780.322,A -85,B 0,C 180,E1 12471.52,E2 12471.52} C_VEL
LIN {X 0,Y 269.954,Z 763.507,A -85,B 0,C 180,E1 12466.746,E2 12466.746} C_VEL
LIN {X 0,Y 281.662,Z 744.596,A -85,B 0,C 180,E1 12462.405,E2 12462.405} C_VEL
LIN {X 0,Y 295.485,Z 724.058,A -85,B 0,C 180,E1 12458.586,E2 12458.586} C_VEL
LIN {X 0,Y 310.184,Z 704.007,A -85,B 0,C 180,E1 12455.582,E2 12455.582} C_VEL
LIN {X 0,Y 295.344,Z 721.305,A -85,B 0,C 180,E1 12452.11,E2 12452.11} C_VEL
LIN {X 0,Y 282.296,Z 737.058,A -85,B 0,C 180,E1 12448.106,E2 12448.106} C_VEL
LIN {X 0,Y 271.599,Z 750.187,A -85,B 0,C 180,E1 12443.891,E2 12443.891} C_VEL
LIN {X 0,Y 262.615,Z 761.402,A -85,B 0,C 180,E1 12439.346,E2 12439.346} C_VEL
LIN {X 0,Y 255.568,Z 770.335,A -85,B 0,C 180,E1 12434.735,E2 12434.735} C_VEL
LIN {X 0,Y 250.054,Z 777.637,A -85,B 0,C 180,E1 12429.903,E2 12429.903} C_VEL
LIN {X 0,Y 245.995,Z 783.332,A -85,B 0,C 180,E1 12424.899,E2 12424.899} C_VEL
LIN {X 0,Y 243.254,Z 787.33,A -85,B 0,C 180,E1 12419.768,E2 12419.768} C_VEL
LIN {X 0,Y 241.685,Z 789.794,A -85,B 0,C 180,E1 12414.543,E2 12414.543} C_VEL
LIN {X 0,Y 240.991,Z 790.711,A -85,B 0,C 180,E1 12409.727,E2 12409.727} C_VEL
LIN {X 0,Y 240.753,Z 790.197,A -85,B 0,C 180,E1 12405.083,E2 12405.083} C_VEL
LIN {X 0,Y 240.754,Z 788.403,A -85,B 0,C 180,E1 12400.346,E2 12400.346} C_VEL
LIN {X 0,Y 241.073,Z 785.385,A -85,B 0,C 180,E1 12395.851,E2 12395.851} C_VEL
LIN {X 0,Y 241.966,Z 780.736,A -85,B 0,C 180,E1 12391.092,E2 12391.092} C_VEL
LIN {X 0,Y 243.662,Z 774.577,A -85,B 0,C 180,E1 12386.365,E2 12386.365} C_VEL
LIN {X 0,Y 246.353,Z 766.481,A -85,B 0,C 180,E1 12381.618,E2 12381.618} C_VEL
LIN {X 0,Y 250.093,Z 756.634,A -85,B 0,C 180,E1 12377.025,E2 12377.025} C_VEL
LIN {X 0,Y 254.674,Z 745.381,A -85,B 0,C 180,E1 12372.769,E2 12372.769} C_VEL
LIN {X 0,Y 260.162,Z 732.3,A -85,B 0,C 180,E1 12368.73,E2 12368.73} C_VEL
LIN {X 0,Y 266.234,Z 717.647,A -85,B 0,C 180,E1 12365.051,E2 12365.051} C_VEL
LIN {X 0,Y 272.419,Z 702.189,A -85,B 0,C 180,E1 12361.852,E2 12361.852} C_VEL
LIN {X 0,Y 279.077,Z 684.732,A -85,B 0,C 180,E1 12358.869,E2 12358.869} C_VEL
LIN {X 0,Y 285.513,Z 666.536,A -85,B 0,C 180,E1 12356.307,E2 12356.307} C_VEL
LIN {X 0,Y 292.09,Z 646.02,A -85,B 0,C 180,E1 12353.95,E2 12353.95} C_VEL
LIN {X 0,Y 297.992,Z 625.126,A -85,B 0,C 180,E1 12352.02,E2 12352.02} C_VEL
LIN {X 0,Y 303.076,Z 604.307,A -85,B 0,C 180,E1 12350.469,E2 12350.469} C_VEL
LIN {X 0,Y 307.674,Z 581.841,A -85,B 0,C 180,E1 12349.142,E2 12349.142} C_VEL
LIN {X 0,Y 311.412,Z 559.137,A -85,B 0,C 180,E1 12348.12,E2 12348.12} C_VEL
LIN {X 0,Y 314.334,Z 535.083,A -85,B 0,C 180,E1 12347.351,E2 12347.351} C_VEL
LIN {X 0,Y 328.234,Z 395.411,A -85,B 0,C 180,E1 12343.747,E2 12343.747} C_VEL
LIN {X 0,Y 317.394,Z 378.662,A -85,B 0,C 180,E1 12340.254,E2 12340.254} C_VEL
LIN {X 0,Y 306.506,Z 362.775,A -85,B 0,C 180,E1 12336.323,E2 12336.323} C_VEL
LIN {X 0,Y 296.027,Z 348.351,A -85,B 0,C 180,E1 12332.034,E2 12332.034} C_VEL
LIN {X 0,Y 287.421,Z 337.113,A -85,B 0,C 180,E1 12328.008,E2 12328.008} C_VEL
LIN {X 0,Y 283.181,Z 331.652,A -85,B 0,C 180,E1 12325.801,E2 12325.801} C_VEL
LIN {X 0,Y 278.929,Z 326.258,A -85,B 0,C 180,E1 12323.415,E2 12323.415} C_VEL
LIN {X 0,Y 275.409,Z 321.615,A -85,B 0,C 180,E1 12321.232,E2 12321.232} C_VEL
LIN {X 0,Y 271.127,Z 316.684,A -85,B 0,C 180,E1 12318.462,E2 12318.462} C_VEL
LIN {X 0,Y 269.973,Z 314.902,A -85,B 0,C 180,E1 12317.598,E2 12317.598} C_VEL
LIN {X 0,Y 266.694,Z 311.592,A -85,B 0,C 180,E1 12315.233,E2 12315.233} C_VEL
LIN {X 0,Y 265.012,Z 308.78,A -85,B 0,C 180,E1 12313.79,E2 12313.79} C_VEL
LIN {X 0,Y 261.696,Z 305.856,A -85,B 0,C 180,E1 12311.052,E2 12311.052} C_VEL
LIN {X 0,Y 259.755,Z 302.428,A -85,B 0,C 180,E1 12309.027,E2 12309.027} C_VEL
LIN {X 0,Y 256.637,Z 300.136,A -85,B 0,C 180,E1 12305.978,E2 12305.978} C_VEL
LIN {X 0,Y 254.797,Z 296.722,A -85,B 0,C 180,E1 12303.429,E2 12303.429} C_VEL
LIN {X 0,Y 254.395,Z 295.942,A -85,B 0,C 180,E1 12302.879,E2 12302.879} C_VEL
LIN {X 0,Y 250.76,Z 293.545,A -85,B 0,C 180,E1 12297.977,E2 12297.977} C_VEL
LIN {X 0,Y 248.925,Z 290.051,A -85,B 0,C 180,E1 12293.956,E2 12293.956} C_VEL
LIN {X 0,Y 248.628,Z 289.254,A -85,B 0,C 180,E1 12293.15,E2 12293.15} C_VEL
LIN {X 0,Y 246.275,Z 288.235,A -85,B 0,C 180,E1 12286.607,E2 12286.607} C_VEL
LIN {X 0,Y 245.399,Z 287.551,A -85,B 0,C 180,E1 12280.009,E2 12280.009} C_VEL
LIN {X 0,Y 245.851,Z 287.921,A -85,B 0,C 180,E1 12273.942,E2 12273.942} C_VEL
LIN {X 0,Y 247.956,Z 289.057,A -85,B 0,C 180,E1 12266.844,E2 12266.844} C_VEL
LIN {X 0,Y 248.801,Z 289.557,A -85,B 0,C 180,E1 12264.955,E2 12264.955} C_VEL
LIN {X 0,Y 250.296,Z 293.034,A -85,B 0,C 180,E1 12261.313,E2 12261.313} C_VEL
LIN {X 0,Y 253.743,Z 295.718,A -85,B 0,C 180,E1 12256.243,E2 12256.243} C_VEL
LIN {X 0,Y 254.583,Z 296.262,A -85,B 0,C 180,E1 12255.194,E2 12255.194} C_VEL
LIN {X 0,Y 256.088,Z 299.533,A -85,B 0,C 180,E1 12252.97,E2 12252.97} C_VEL
LIN {X 0,Y 259.379,Z 302.282,A -85,B 0,C 180,E1 12249.538,E2 12249.538} C_VEL
LIN {X 0,Y 260.16,Z 303.069,A -85,B 0,C 180,E1 12248.784,E2 12248.784} C_VEL
LIN {X 0,Y 262.386,Z 306.753,A -85,B 0,C 180,E1 12246.451,E2 12246.451} C_VEL
LIN {X 0,Y 265.416,Z 309.3,A -85,B 0,C 180,E1 12243.993,E2 12243.993} C_VEL
LIN {X 0,Y 268.09,Z 313.394,A -85,B 0,C 180,E1 12241.707,E2 12241.707} C_VEL
LIN {X 0,Y 270.601,Z 315.721,A -85,B 0,C 180,E1 12239.944,E2 12239.944} C_VEL
LIN {X 0,Y 271.199,Z 316.787,A -85,B 0,C 180,E1 12239.475,E2 12239.475} C_VEL
LIN {X 0,Y 273.111,Z 321.295,A -85,B 0,C 180,E1 12237.91,E2 12237.91} C_VEL
LIN {X 0,Y 276.899,Z 333.514,A -85,B 0,C 180,E1 12234.669,E2 12234.669} C_VEL
LIN {X 0,Y 278.658,Z 336.647,A -85,B 0,C 180,E1 12233.51,E2 12233.51} C_VEL
LIN {X 0,Y 284.386,Z 344.667,A -85,B 0,C 180,E1 12230.282,E2 12230.282} C_VEL
LIN {X 0,Y 291.599,Z 355.245,A -85,B 0,C 180,E1 12226.615,E2 12226.615} C_VEL
LIN {X 0,Y 299.916,Z 367.749,A -85,B 0,C 180,E1 12222.838,E2 12222.838} C_VEL
LIN {X 0,Y 308.872,Z 382.027,A -85,B 0,C 180,E1 12219.188,E2 12219.188} C_VEL
LIN {X 0,Y 318.035,Z 397.293,A -85,B 0,C 180,E1 12215.825,E2 12215.825} C_VEL
LIN {X 0,Y 325.328,Z 410.398,A -85,B 0,C 180,E1 12213.347,E2 12213.347} C_VEL
LIN {X 0,Y 305.981,Z 592.918,A -85,B 0,C 180,E1 12208.532,E2 12208.532} C_VEL
LIN {X 0,Y 302.084,Z 616.69,A -85,B 0,C 180,E1 12207.639,E2 12207.639} C_VEL
LIN {X 0,Y 297.196,Z 639.233,A -85,B 0,C 180,E1 12206.511,E2 12206.511} C_VEL
LIN {X 0,Y 291.516,Z 661.364,A -85,B 0,C 180,E1 12205.054,E2 12205.054} C_VEL
LIN {X 0,Y 285.144,Z 682.901,A -85,B 0,C 180,E1 12203.244,E2 12203.244} C_VEL
LIN {X 0,Y 278.56,Z 702.809,A -85,B 0,C 180,E1 12201.155,E2 12201.155} C_VEL
LIN {X 0,Y 271.367,Z 722.68,A -85,B 0,C 180,E1 12198.569,E2 12198.569} C_VEL
LIN {X 0,Y 264.315,Z 740.807,A -85,B 0,C 180,E1 12195.636,E2 12195.636} C_VEL
LIN {X 0,Y 257.605,Z 757.209,A -85,B 0,C 180,E1 12192.393,E2 12192.393} C_VEL
LIN {X 0,Y 251.209,Z 772.629,A -85,B 0,C 180,E1 12188.671,E2 12188.671} C_VEL
LIN {X 0,Y 245.662,Z 786.136,A -85,B 0,C 180,E1 12184.696,E2 12184.696} C_VEL
LIN {X 0,Y 240.873,Z 798.272,A -85,B 0,C 180,E1 12180.295,E2 12180.295} C_VEL
LIN {X 0,Y 237.226,Z 808.447,A -85,B 0,C 180,E1 12175.727,E2 12175.727} C_VEL
LIN {X 0,Y 234.574,Z 817.369,A -85,B 0,C 180,E1 12170.716,E2 12170.716} C_VEL
LIN {X 0,Y 233.149,Z 824.023,A -85,B 0,C 180,E1 12165.927,E2 12165.927} C_VEL
LIN {X 0,Y 232.61,Z 828.843,A -85,B 0,C 180,E1 12161.15,E2 12161.15} C_VEL
LIN {X 0,Y 232.635,Z 832.118,A -85,B 0,C 180,E1 12156.414,E2 12156.414} C_VEL
LIN {X 0,Y 232.779,Z 833.588,A -85,B 0,C 180,E1 12152.213,E2 12152.213} C_VEL
LIN {X 0,Y 232.77,Z 833.844,A -85,B 0,C 180,E1 12148.275,E2 12148.275} C_VEL
LIN {X 0,Y 232.581,Z 832.777,A -85,B 0,C 180,E1 12143.828,E2 12143.828} C_VEL
LIN {X 0,Y 232.511,Z 830.3,A -85,B 0,C 180,E1 12139.342,E2 12139.342} C_VEL
LIN {X 0,Y 233.058,Z 825.788,A -85,B 0,C 180,E1 12134.061,E2 12134.061} C_VEL
LIN {X 0,Y 234.656,Z 819.687,A -85,B 0,C 180,E1 12128.936,E2 12128.936} C_VEL
LIN {X 0,Y 237.792,Z 811.312,A -85,B 0,C 180,E1 12123.529,E2 12123.529} C_VEL
LIN {X 0,Y 242.909,Z 800.423,A -85,B 0,C 180,E1 12117.991,E2 12117.991} C_VEL
LIN {X 0,Y 249.48,Z 788.401,A -85,B 0,C 180,E1 12113.044,E2 12113.044} C_VEL
LIN {X 0,Y 258.581,Z 773.225,A -85,B 0,C 180,E1 12108.012,E2 12108.012} C_VEL
LIN {X 0,Y 270.613,Z 754.913,A -85,B 0,C 180,E1 12103.123,E2 12103.123} C_VEL
LIN {X 0,Y 285.65,Z 734.099,A -85,B 0,C 180,E1 12098.686,E2 12098.686} C_VEL
LIN {X 0,Y 300.786,Z 715.019,A -85,B 0,C 180,E1 12095.429,E2 12095.429} C_VEL
LIN {X 0,Y 285.436,Z 731.253,A -85,B 0,C 180,E1 12091.7,E2 12091.7} C_VEL
LIN {X 0,Y 271.972,Z 746.026,A -85,B 0,C 180,E1 12087.36,E2 12087.36} C_VEL
LIN {X 0,Y 260.625,Z 758.735,A -85,B 0,C 180,E1 12082.562,E2 12082.562} C_VEL
LIN {X 0,Y 251.337,Z 769.329,A -85,B 0,C 180,E1 12077.362,E2 12077.362} C_VEL
LIN {X 0,Y 244.339,Z 777.512,A -85,B 0,C 180,E1 12072.049,E2 12072.049} C_VEL
LIN {X 0,Y 239.356,Z 783.56,A -85,B 0,C 180,E1 12066.72,E2 12066.72} C_VEL
LIN {X 0,Y 235.963,Z 787.91,A -85,B 0,C 180,E1 12061.217,E2 12061.217} C_VEL
LIN {X 0,Y 234.052,Z 790.512,A -85,B 0,C 180,E1 12055.839,E2 12055.839} C_VEL
LIN {X 0,Y 233.153,Z 791.528,A -85,B 0,C 180,E1 12050.874,E2 12050.874} C_VEL
LIN {X 0,Y 232.817,Z 791.169,A -85,B 0,C 180,E1 12046.075,E2 12046.075} C_VEL
LIN {X 0,Y 232.76,Z 789.692,A -85,B 0,C 180,E1 12041.469,E2 12041.469} C_VEL
LIN {X 0,Y 233.006,Z 786.781,A -85,B 0,C 180,E1 12036.683,E2 12036.683} C_VEL
LIN {X 0,Y 233.842,Z 782.305,A -85,B 0,C 180,E1 12031.67,E2 12031.67} C_VEL
LIN {X 0,Y 235.472,Z 776.282,A -85,B 0,C 180,E1 12026.775,E2 12026.775} C_VEL
LIN {X 0,Y 238.115,Z 768.469,A -85,B 0,C 180,E1 12021.889,E2 12021.889} C_VEL
LIN {X 0,Y 241.967,Z 758.627,A -85,B 0,C 180,E1 12017.02,E2 12017.02} C_VEL
LIN {X 0,Y 246.636,Z 747.572,A -85,B 0,C 180,E1 12012.613,E2 12012.613} C_VEL
LIN {X 0,Y 252.14,Z 734.82,A -85,B 0,C 180,E1 12008.507,E2 12008.507} C_VEL
LIN {X 0,Y 258.154,Z 720.815,A -85,B 0,C 180,E1 12004.812,E2 12004.812} C_VEL
LIN {X 0,Y 265.077,Z 704.208,A -85,B 0,C 180,E1 12001.221,E2 12001.221} C_VEL
LIN {X 0,Y 271.891,Z 687.02,A -85,B 0,C 180,E1 11998.185,E2 11998.185} C_VEL
LIN {X 0,Y 278.695,Z 668.514,A -85,B 0,C 180,E1 11995.502,E2 11995.502} C_VEL
LIN {X 0,Y 285.46,Z 648.065,A -85,B 0,C 180,E1 11993.099,E2 11993.099} C_VEL
LIN {X 0,Y 291.245,Z 628.429,A -85,B 0,C 180,E1 11991.227,E2 11991.227} C_VEL
LIN {X 0,Y 296.985,Z 606.032,A -85,B 0,C 180,E1 11989.506,E2 11989.506} C_VEL
LIN {X 0,Y 301.602,Z 584.565,A -85,B 0,C 180,E1 11988.201,E2 11988.201} C_VEL
LIN {X 0,Y 305.618,Z 561.392,A -85,B 0,C 180,E1 11987.121,E2 11987.121} C_VEL
LIN {X 0,Y 308.693,Z 537.148,A -85,B 0,C 180,E1 11986.323,E2 11986.323} C_VEL
LIN {X 0,Y 322.916,Z 399.246,A -85,B 0,C 180,E1 11982.726,E2 11982.726} C_VEL
LIN {X 0,Y 311.84,Z 382.172,A -85,B 0,C 180,E1 11979.01,E2 11979.01} C_VEL
LIN {X 0,Y 302.237,Z 368.19,A -85,B 0,C 180,E1 11975.412,E2 11975.412} C_VEL
LIN {X 0,Y 293.123,Z 355.405,A -85,B 0,C 180,E1 11971.566,E2 11971.566} C_VEL
LIN {X 0,Y 284.665,Z 344.246,A -85,B 0,C 180,E1 11967.536,E2 11967.536} C_VEL
LIN {X 0,Y 280.441,Z 338.701,A -85,B 0,C 180,E1 11965.247,E2 11965.247} C_VEL
LIN {X 0,Y 276.231,Z 333.372,A -85,B 0,C 180,E1 11962.87,E2 11962.87} C_VEL
LIN {X 0,Y 272.136,Z 328.051,A -85,B 0,C 180,E1 11960.272,E2 11960.272} C_VEL
LIN {X 0,Y 268.648,Z 323.846,A -85,B 0,C 180,E1 11957.918,E2 11957.918} C_VEL
LIN {X 0,Y 267.506,Z 322.226,A -85,B 0,C 180,E1 11957.043,E2 11957.043} C_VEL
LIN {X 0,Y 264.096,Z 318.492,A -85,B 0,C 180,E1 11954.522,E2 11954.522} C_VEL
LIN {X 0,Y 262.874,Z 316.369,A -85,B 0,C 180,E1 11953.421,E2 11953.421} C_VEL
LIN {X 0,Y 259.425,Z 313.173,A -85,B 0,C 180,E1 11950.528,E2 11950.528} C_VEL
LIN {X 0,Y 257.656,Z 310.052,A -85,B 0,C 180,E1 11948.609,E2 11948.609} C_VEL
LIN {X 0,Y 254.557,Z 307.614,A -85,B 0,C 180,E1 11945.522,E2 11945.522} C_VEL
LIN {X 0,Y 252.681,Z 304.085,A -85,B 0,C 180,E1 11942.905,E2 11942.905} C_VEL
LIN {X 0,Y 251.769,Z 303.387,A -85,B 0,C 180,E1 11941.8,E2 11941.8} C_VEL
LIN {X 0,Y 248.815,Z 301.13,A -85,B 0,C 180,E1 11937.544,E2 11937.544} C_VEL
LIN {X 0,Y 247.079,Z 297.749,A -85,B 0,C 180,E1 11933.632,E2 11933.632} C_VEL
LIN {X 0,Y 246.812,Z 297.037,A -85,B 0,C 180,E1 11932.874,E2 11932.874} C_VEL
LIN {X 0,Y 244.459,Z 295.972,A -85,B 0,C 180,E1 11925.952,E2 11925.952} C_VEL
LIN {X 0,Y 243.706,Z 295.373,A -85,B 0,C 180,E1 11919.788,E2 11919.788} C_VEL
LIN {X 0,Y 244.249,Z 295.819,A -85,B 0,C 180,E1 11913.543,E2 11913.543} C_VEL
LIN {X 0,Y 246.421,Z 296.922,A -85,B 0,C 180,E1 11906.504,E2 11906.504} C_VEL
LIN {X 0,Y 246.962,Z 297.259,A -85,B 0,C 180,E1 11905.282,E2 11905.282} C_VEL
LIN {X 0,Y 248.647,Z 300.995,A -85,B 0,C 180,E1 11901.214,E2 11901.214} C_VEL
LIN {X 0,Y 252.178,Z 303.589,A -85,B 0,C 180,E1 11896.11,E2 11896.11} C_VEL
LIN {X 0,Y 252.688,Z 304.156,A -85,B 0,C 180,E1 11895.429,E2 11895.429} C_VEL
LIN {X 0,Y 254.294,Z 307.388,A -85,B 0,C 180,E1 11893.063,E2 11893.063} C_VEL
LIN {X 0,Y 257.621,Z 310.085,A -85,B 0,C 180,E1 11889.604,E2 11889.604} C_VEL
LIN {X 0,Y 260.764,Z 314.816,A -85,B 0,C 180,E1 11886.381,E2 11886.381} C_VEL
LIN {X 0,Y 263.217,Z 316.92,A -85,B 0,C 180,E1 11884.354,E2 11884.354} C_VEL
LIN {X 0,Y 266.083,Z 321.085,A -85,B 0,C 180,E1 11881.935,E2 11881.935} C_VEL
LIN {X 0,Y 268.259,Z 323.162,A -85,B 0,C 180,E1 11880.371,E2 11880.371} C_VEL
LIN {X 0,Y 271.553,Z 327.568,A -85,B 0,C 180,E1 11877.993,E2 11877.993} C_VEL
LIN {X 0,Y 273.22,Z 329.404,A -85,B 0,C 180,E1 11876.903,E2 11876.903} C_VEL
LIN {X 0,Y 278.658,Z 336.647,A -85,B 0,C 180,E1 11873.51,E2 11873.51} C_VEL
LIN {X 0,Y 280.434,Z 339.996,A -85,B 0,C 180,E1 11872.391,E2 11872.391} C_VEL
LIN {X 0,Y 282.608,Z 347.591,A -85,B 0,C 180,E1 11870.779,E2 11870.779} C_VEL
LIN {X 0,Y 285.022,Z 356.096,A -85,B 0,C 180,E1 11869.028,E2 11869.028} C_VEL
LIN {X 0,Y 286.643,Z 359.087,A -85,B 0,C 180,E1 11868.14,E2 11868.14} C_VEL
LIN {X 0,Y 295.902,Z 373.115,A -85,B 0,C 180,E1 11863.761,E2 11863.761} C_VEL
LIN {X 0,Y 305.267,Z 388.281,A -85,B 0,C 180,E1 11859.832,E2 11859.832} C_VEL
LIN {X 0,Y 314.247,Z 403.398,A -85,B 0,C 180,E1 11856.463,E2 11856.463} C_VEL
LIN {X 0,Y 320.115,Z 414.212,A -85,B 0,C 180,E1 11854.39,E2 11854.39} C_VEL
LIN {X 0,Y 300.563,Z 592.368,A -85,B 0,C 180,E1 11849.65,E2 11849.65} C_VEL
LIN {X 0,Y 296.566,Z 616.091,A -85,B 0,C 180,E1 11848.752,E2 11848.752} C_VEL
LIN {X 0,Y 291.593,Z 638.384,A -85,B 0,C 180,E1 11847.633,E2 11847.633} C_VEL
LIN {X 0,Y 285.805,Z 660.36,A -85,B 0,C 180,E1 11846.184,E2 11846.184} C_VEL
LIN {X 0,Y 279.254,Z 681.958,A -85,B 0,C 180,E1 11844.362,E2 11844.362} C_VEL
LIN {X 0,Y 272.464,Z 701.921,A -85,B 0,C 180,E1 11842.258,E2 11842.258} C_VEL
LIN {X 0,Y 265.029,Z 721.815,A -85,B 0,C 180,E1 11839.643,E2 11839.643} C_VEL
LIN {X 0,Y 257.966,Z 739.38,A -85,B 0,C 180,E1 11836.771,E2 11836.771} C_VEL
LIN {X 0,Y 251.095,Z 755.626,A -85,B 0,C 180,E1 11833.538,E2 11833.538} C_VEL
LIN {X 0,Y 244.659,Z 770.6,A -85,B 0,C 180,E1 11829.909,E2 11829.909} C_VEL
LIN {X 0,Y 238.81,Z 784.205,A -85,B 0,C 180,E1 11825.881,E2 11825.881} C_VEL
LIN {X 0,Y 233.771,Z 796.31,A -85,B 0,C 180,E1 11821.45,E2 11821.45} C_VEL
LIN {X 0,Y 229.732,Z 806.975,A -85,B 0,C 180,E1 11816.631,E2 11816.631} C_VEL
LIN {X 0,Y 226.958,Z 815.691,A -85,B 0,C 180,E1 11811.716,E2 11811.716} C_VEL
LIN {X 0,Y 225.403,Z 822.168,A -85,B 0,C 180,E1 11807.021,E2 11807.021} C_VEL
LIN {X 0,Y 224.675,Z 827.574,A -85,B 0,C 180,E1 11801.81,E2 11801.81} C_VEL
LIN {X 0,Y 224.639,Z 830.725,A -85,B 0,C 180,E1 11797.414,E2 11797.414} C_VEL
LIN {X 0,Y 224.806,Z 832.617,A -85,B 0,C 180,E1 11792.802,E2 11792.802} C_VEL
LIN {X 0,Y 224.832,Z 833.042,A -85,B 0,C 180,E1 11788.978,E2 11788.978} C_VEL
LIN {X 0,Y 224.667,Z 832.422,A -85,B 0,C 180,E1 11784.891,E2 11784.891} C_VEL
LIN {X 0,Y 224.511,Z 830.278,A -85,B 0,C 180,E1 11779.995,E2 11779.995} C_VEL
LIN {X 0,Y 224.878,Z 826.599,A -85,B 0,C 180,E1 11775.053,E2 11775.053} C_VEL
LIN {X 0,Y 226.411,Z 820.734,A -85,B 0,C 180,E1 11769.432,E2 11769.432} C_VEL
LIN {X 0,Y 229.262,Z 813.455,A -85,B 0,C 180,E1 11764.141,E2 11764.141} C_VEL
LIN {X 0,Y 234.058,Z 803.726,A -85,B 0,C 180,E1 11758.587,E2 11758.587} C_VEL
LIN {X 0,Y 241.119,Z 791.535,A -85,B 0,C 180,E1 11753.036,E2 11753.036} C_VEL
LIN {X 0,Y 250.332,Z 777.401,A -85,B 0,C 180,E1 11747.852,E2 11747.852} C_VEL
LIN {X 0,Y 262.784,Z 759.996,A -85,B 0,C 180,E1 11742.746,E2 11742.746} C_VEL
LIN {X 0,Y 278.408,Z 740.191,A -85,B 0,C 180,E1 11738.138,E2 11738.138} C_VEL
LIN {X 0,Y 291.285,Z 725.217,A -85,B 0,C 180,E1 11735.279,E2 11735.279} C_VEL
LIN {X 0,Y 275.455,Z 740.419,A -85,B 0,C 180,E1 11731.272,E2 11731.272} C_VEL
LIN {X 0,Y 261.555,Z 754.273,A -85,B 0,C 180,E1 11726.549,E2 11726.549} C_VEL
LIN {X 0,Y 250.046,Z 765.938,A -85,B 0,C 180,E1 11721.341,E2 11721.341} C_VEL
LIN {X 0,Y 241.12,Z 775.211,A -85,B 0,C 180,E1 11715.887,E2 11715.887} C_VEL
LIN {X 0,Y 234.539,Z 782.217,A -85,B 0,C 180,E1 11710.317,E2 11710.317} C_VEL
LIN {X 0,Y 230.171,Z 787,A -85,B 0,C 180,E1 11704.987,E2 11704.987} C_VEL
LIN {X 0,Y 227.196,Z 790.423,A -85,B 0,C 180,E1 11699.247,E2 11699.247} C_VEL
LIN {X 0,Y 225.675,Z 792.143,A -85,B 0,C 180,E1 11693.9,E2 11693.9} C_VEL
LIN {X 0,Y 225.01,Z 792.356,A -85,B 0,C 180,E1 11688.988,E2 11688.988} C_VEL
LIN {X 0,Y 224.795,Z 791.352,A -85,B 0,C 180,E1 11683.898,E2 11683.898} C_VEL
LIN {X 0,Y 224.855,Z 789.159,A -85,B 0,C 180,E1 11679.166,E2 11679.166} C_VEL
LIN {X 0,Y 225.405,Z 785.328,A -85,B 0,C 180,E1 11673.955,E2 11673.955} C_VEL
LIN {X 0,Y 226.681,Z 780.057,A -85,B 0,C 180,E1 11668.841,E2 11668.841} C_VEL
LIN {X 0,Y 228.875,Z 773.156,A -85,B 0,C 180,E1 11663.865,E2 11663.865} C_VEL
LIN {X 0,Y 232.29,Z 764.26,A -85,B 0,C 180,E1 11658.815,E2 11658.815} C_VEL
LIN {X 0,Y 236.707,Z 753.881,A -85,B 0,C 180,E1 11654.109,E2 11654.109} C_VEL
LIN {X 0,Y 241.969,Z 742.074,A -85,B 0,C 180,E1 11649.78,E2 11649.78} C_VEL
LIN {X 0,Y 248.001,Z 728.605,A -85,B 0,C 180,E1 11645.777,E2 11645.777} C_VEL
LIN {X 0,Y 254.756,Z 713.244,A -85,B 0,C 180,E1 11642.04,E2 11642.04} C_VEL
LIN {X 0,Y 261.654,Z 696.904,A -85,B 0,C 180,E1 11638.784,E2 11638.784} C_VEL
LIN {X 0,Y 268.555,Z 679.492,A -85,B 0,C 180,E1 11635.93,E2 11635.93} C_VEL
LIN {X 0,Y 275.532,Z 660.197,A -85,B 0,C 180,E1 11633.361,E2 11633.361} C_VEL
LIN {X 0,Y 282.023,Z 640.242,A -85,B 0,C 180,E1 11631.197,E2 11631.197} C_VEL
LIN {X 0,Y 288.16,Z 618.793,A -85,B 0,C 180,E1 11629.315,E2 11629.315} C_VEL
LIN {X 0,Y 293.445,Z 597.214,A -85,B 0,C 180,E1 11627.805,E2 11627.805} C_VEL
LIN {X 0,Y 298.086,Z 574.285,A -85,B 0,C 180,E1 11626.557,E2 11626.557} C_VEL
LIN {X 0,Y 301.813,Z 550.442,A -85,B 0,C 180,E1 11625.603,E2 11625.603} C_VEL
LIN {X 0,Y 309.063,Z 483.535,A -85,B 0,C 180,E1 11623.778,E2 11623.778} C_VEL
LIN {X 0,Y 317.706,Z 403.165,A -85,B 0,C 180,E1 11621.667,E2 11621.667} C_VEL
LIN {X 0,Y 306.466,Z 385.761,A -85,B 0,C 180,E1 11617.736,E2 11617.736} C_VEL
LIN {X 0,Y 296.526,Z 371.319,A -85,B 0,C 180,E1 11613.825,E2 11613.825} C_VEL
LIN {X 0,Y 288.101,Z 359.718,A -85,B 0,C 180,E1 11610.091,E2 11610.091} C_VEL
LIN {X 0,Y 281.75,Z 351.152,A -85,B 0,C 180,E1 11606.951,E2 11606.951} C_VEL
LIN {X 0,Y 277.733,Z 345.819,A -85,B 0,C 180,E1 11604.735,E2 11604.735} C_VEL
LIN {X 0,Y 273.598,Z 340.52,A -85,B 0,C 180,E1 11602.337,E2 11602.337} C_VEL
LIN {X 0,Y 269.541,Z 335.279,A -85,B 0,C 180,E1 11599.746,E2 11599.746} C_VEL
LIN {X 0,Y 266.034,Z 330.745,A -85,B 0,C 180,E1 11597.246,E2 11597.246} C_VEL
LIN {X 0,Y 261.531,Z 325.371,A -85,B 0,C 180,E1 11593.797,E2 11593.797} C_VEL
LIN {X 0,Y 260.516,Z 323.792,A -85,B 0,C 180,E1 11592.859,E2 11592.859} C_VEL
LIN {X 0,Y 256.925,Z 320.106,A -85,B 0,C 180,E1 11589.738,E2 11589.738} C_VEL
LIN {X 0,Y 255.561,Z 317.662,A -85,B 0,C 180,E1 11588.183,E2 11588.183} C_VEL
LIN {X 0,Y 252.385,Z 314.945,A -85,B 0,C 180,E1 11584.922,E2 11584.922} C_VEL
LIN {X 0,Y 250.4,Z 311.343,A -85,B 0,C 180,E1 11582.151,E2 11582.151} C_VEL
LIN {X 0,Y 247.218,Z 309.118,A -85,B 0,C 180,E1 11577.695,E2 11577.695} C_VEL
LIN {X 0,Y 245.231,Z 305.383,A -85,B 0,C 180,E1 11573.26,E2 11573.26} C_VEL
LIN {X 0,Y 244.982,Z 304.812,A -85,B 0,C 180,E1 11572.55,E2 11572.55} C_VEL
LIN {X 0,Y 242.643,Z 303.71,A -85,B 0,C 180,E1 11565.464,E2 11565.464} C_VEL
LIN {X 0,Y 242.014,Z 303.199,A -85,B 0,C 180,E1 11559.419,E2 11559.419} C_VEL
LIN {X 0,Y 242.706,Z 303.757,A -85,B 0,C 180,E1 11552.937,E2 11552.937} C_VEL
LIN {X 0,Y 245.087,Z 304.84,A -85,B 0,C 180,E1 11545.748,E2 11545.748} C_VEL
LIN {X 0,Y 246.848,Z 308.762,A -85,B 0,C 180,E1 11541.376,E2 11541.376} C_VEL
LIN {X 0,Y 250.507,Z 311.417,A -85,B 0,C 180,E1 11536.101,E2 11536.101} C_VEL
LIN {X 0,Y 252.4,Z 315.112,A -85,B 0,C 180,E1 11533.28,E2 11533.28} C_VEL
LIN {X 0,Y 255.925,Z 318.251,A -85,B 0,C 180,E1 11529.554,E2 11529.554} C_VEL
LIN {X 0,Y 258.722,Z 322.407,A -85,B 0,C 180,E1 11526.709,E2 11526.709} C_VEL
LIN {X 0,Y 261.032,Z 324.522,A -85,B 0,C 180,E1 11524.721,E2 11524.721} C_VEL
LIN {X 0,Y 264.081,Z 328.772,A -85,B 0,C 180,E1 11522.167,E2 11522.167} C_VEL
LIN {X 0,Y 265.972,Z 330.685,A -85,B 0,C 180,E1 11520.759,E2 11520.759} C_VEL
LIN {X 0,Y 269.407,Z 335.143,A -85,B 0,C 180,E1 11518.296,E2 11518.296} C_VEL
LIN {X 0,Y 270.942,Z 337.002,A -85,B 0,C 180,E1 11517.247,E2 11517.247} C_VEL
LIN {X 0,Y 277.234,Z 345.291,A -85,B 0,C 180,E1 11513.318,E2 11513.318} C_VEL
LIN {X 0,Y 284.746,Z 356.297,A -85,B 0,C 180,E1 11509.118,E2 11509.118} C_VEL
LIN {X 0,Y 286.643,Z 359.087,A -85,B 0,C 180,E1 11508.14,E2 11508.14} C_VEL
LIN {X 0,Y 288.584,Z 362.821,A -85,B 0,C 180,E1 11507.116,E2 11507.116} C_VEL
LIN {X 0,Y 290.829,Z 370.977,A -85,B 0,C 180,E1 11505.669,E2 11505.669} C_VEL
LIN {X 0,Y 293.335,Z 380.179,A -85,B 0,C 180,E1 11504.112,E2 11504.112} C_VEL
LIN {X 0,Y 295.018,Z 383.579,A -85,B 0,C 180,E1 11503.31,E2 11503.31} C_VEL
LIN {X 0,Y 304.055,Z 398.451,A -85,B 0,C 180,E1 11499.548,E2 11499.548} C_VEL
LIN {X 0,Y 313.84,Z 415.545,A -85,B 0,C 180,E1 11495.882,E2 11495.882} C_VEL
LIN {X 0,Y 314.977,Z 417.987,A -85,B 0,C 180,E1 11495.463,E2 11495.463} C_VEL
LIN {X 0,Y 295.224,Z 591.236,A -85,B 0,C 180,E1 11490.807,E2 11490.807} C_VEL
LIN {X 0,Y 291.14,Z 614.958,A -85,B 0,C 180,E1 11489.905,E2 11489.905} C_VEL
LIN {X 0,Y 285.974,Z 637.597,A -85,B 0,C 180,E1 11488.771,E2 11488.771} C_VEL
LIN {X 0,Y 279.932,Z 659.928,A -85,B 0,C 180,E1 11487.29,E2 11487.29} C_VEL
LIN {X 0,Y 273.08,Z 681.848,A -85,B 0,C 180,E1 11485.42,E2 11485.42} C_VEL
LIN {X 0,Y 266.209,Z 701.44,A -85,B 0,C 180,E1 11483.328,E2 11483.328} C_VEL
LIN {X 0,Y 258.511,Z 721.418,A -85,B 0,C 180,E1 11480.67,E2 11480.67} C_VEL
LIN {X 0,Y 251.112,Z 739.234,A -85,B 0,C 180,E1 11477.705,E2 11477.705} C_VEL
LIN {X 0,Y 243.889,Z 755.714,A -85,B 0,C 180,E1 11474.342,E2 11474.342} C_VEL
LIN {X 0,Y 237.051,Z 771.018,A -85,B 0,C 180,E1 11470.504,E2 11470.504} C_VEL
LIN {X 0,Y 231.039,Z 784.509,A -85,B 0,C 180,E1 11466.359,E2 11466.359} C_VEL
LIN {X 0,Y 225.864,Z 796.493,A -85,B 0,C 180,E1 11461.785,E2 11461.785} C_VEL
LIN {X 0,Y 221.916,Z 806.493,A -85,B 0,C 180,E1 11457.066,E2 11457.066} C_VEL
LIN {X 0,Y 219.036,Z 815.162,A -85,B 0,C 180,E1 11451.979,E2 11451.979} C_VEL
LIN {X 0,Y 217.388,Z 821.84,A -85,B 0,C 180,E1 11446.919,E2 11446.919} C_VEL
LIN {X 0,Y 216.702,Z 826.937,A -85,B 0,C 180,E1 11441.711,E2 11441.711} C_VEL
LIN {X 0,Y 216.689,Z 830.038,A -85,B 0,C 180,E1 11437.154,E2 11437.154} C_VEL
LIN {X 0,Y 216.857,Z 831.785,A -85,B 0,C 180,E1 11432.64,E2 11432.64} C_VEL
LIN {X 0,Y 216.867,Z 832.205,A -85,B 0,C 180,E1 11428.676,E2 11428.676} C_VEL
LIN {X 0,Y 216.688,Z 831.633,A -85,B 0,C 180,E1 11424.702,E2 11424.702} C_VEL
LIN {X 0,Y 216.526,Z 829.738,A -85,B 0,C 180,E1 11419.891,E2 11419.891} C_VEL
LIN {X 0,Y 216.981,Z 825.895,A -85,B 0,C 180,E1 11414.391,E2 11414.391} C_VEL
LIN {X 0,Y 218.734,Z 820.118,A -85,B 0,C 180,E1 11408.548,E2 11408.548} C_VEL
LIN {X 0,Y 222,Z 812.725,A -85,B 0,C 180,E1 11402.94,E2 11402.94} C_VEL
LIN {X 0,Y 227.436,Z 802.916,A -85,B 0,C 180,E1 11397.11,E2 11397.11} C_VEL
LIN {X 0,Y 235.146,Z 791.051,A -85,B 0,C 180,E1 11391.483,E2 11391.483} C_VEL
LIN {X 0,Y 245.834,Z 776.346,A -85,B 0,C 180,E1 11385.931,E2 11385.931} C_VEL
LIN {X 0,Y 260.46,Z 758.202,A -85,B 0,C 180,E1 11380.526,E2 11380.526} C_VEL
LIN {X 0,Y 277.284,Z 739.356,A -85,B 0,C 180,E1 11376.124,E2 11376.124} C_VEL
LIN {X 0,Y 281.807,Z 734.56,A -85,B 0,C 180,E1 11375.155,E2 11375.155} C_VEL
LIN {X 0,Y 265.403,Z 748.863,A -85,B 0,C 180,E1 11370.823,E2 11370.823} C_VEL
LIN {X 0,Y 251.156,Z 761.713,A -85,B 0,C 180,E1 11365.72,E2 11365.72} C_VEL
LIN {X 0,Y 239.858,Z 772.07,A -85,B 0,C 180,E1 11360.245,E2 11360.245} C_VEL
LIN {X 0,Y 231.255,Z 780.176,A -85,B 0,C 180,E1 11354.526,E2 11354.526} C_VEL
LIN {X 0,Y 224.84,Z 786.33,A -85,B 0,C 180,E1 11348.442,E2 11348.442} C_VEL
LIN {X 0,Y 220.792,Z 790.271,A -85,B 0,C 180,E1 11342.599,E2 11342.599} C_VEL
LIN {X 0,Y 218.448,Z 792.543,A -85,B 0,C 180,E1 11336.855,E2 11336.855} C_VEL
LIN {X 0,Y 217.299,Z 793.343,A -85,B 0,C 180,E1 11331.27,E2 11331.27} C_VEL
LIN {X 0,Y 216.89,Z 792.694,A -85,B 0,C 180,E1 11326.134,E2 11326.134} C_VEL
LIN {X 0,Y 216.83,Z 790.804,A -85,B 0,C 180,E1 11320.893,E2 11320.893} C_VEL
LIN {X 0,Y 217.12,Z 787.828,A -85,B 0,C 180,E1 11316.098,E2 11316.098} C_VEL
LIN {X 0,Y 218.136,Z 782.944,A -85,B 0,C 180,E1 11310.635,E2 11310.635} C_VEL
LIN {X 0,Y 220.07,Z 776.666,A -85,B 0,C 180,E1 11305.4,E2 11305.4} C_VEL
LIN {X 0,Y 223.165,Z 768.438,A -85,B 0,C 180,E1 11300.162,E2 11300.162} C_VEL
LIN {X 0,Y 227.31,Z 758.737,A -85,B 0,C 180,E1 11295.275,E2 11295.275} C_VEL
LIN {X 0,Y 232.696,Z 746.944,A -85,B 0,C 180,E1 11290.495,E2 11290.495} C_VEL
LIN {X 0,Y 238.504,Z 734.555,A -85,B 0,C 180,E1 11286.407,E2 11286.407} C_VEL
LIN {X 0,Y 245.286,Z 719.787,A -85,B 0,C 180,E1 11282.465,E2 11282.465} C_VEL
LIN {X 0,Y 252.273,Z 703.982,A -85,B 0,C 180,E1 11279.021,E2 11279.021} C_VEL
LIN {X 0,Y 259.94,Z 685.624,A -85,B 0,C 180,E1 11275.765,E2 11275.765} C_VEL
LIN {X 0,Y 266.855,Z 667.697,A -85,B 0,C 180,E1 11273.169,E2 11273.169} C_VEL
LIN {X 0,Y 273.818,Z 647.811,A -85,B 0,C 180,E1 11270.817,E2 11270.817} C_VEL
LIN {X 0,Y 280.291,Z 626.801,A -85,B 0,C 180,E1 11268.824,E2 11268.824} C_VEL
LIN {X 0,Y 285.792,Z 606.131,A -85,B 0,C 180,E1 11267.247,E2 11267.247} C_VEL
LIN {X 0,Y 290.991,Z 582.778,A -85,B 0,C 180,E1 11265.841,E2 11265.841} C_VEL
LIN {X 0,Y 295.083,Z 559.814,A -85,B 0,C 180,E1 11264.796,E2 11264.796} C_VEL
LIN {X 0,Y 298.281,Z 535.758,A -85,B 0,C 180,E1 11264.015,E2 11264.015} C_VEL
LIN {X 0,Y 312.562,Z 407.248,A -85,B 0,C 180,E1 11260.601,E2 11260.601} C_VEL
LIN {X 0,Y 302.442,Z 391.456,A -85,B 0,C 180,E1 11256.932,E2 11256.932} C_VEL
LIN {X 0,Y 293.197,Z 377.826,A -85,B 0,C 180,E1 11253.179,E2 11253.179} C_VEL
LIN {X 0,Y 285.103,Z 366.5,A -85,B 0,C 180,E1 11249.49,E2 11249.49} C_VEL
LIN {X 0,Y 278.472,Z 357.549,A -85,B 0,C 180,E1 11246.137,E2 11246.137} C_VEL
LIN {X 0,Y 274.78,Z 352.681,A -85,B 0,C 180,E1 11244.102,E2 11244.102} C_VEL
LIN {X 0,Y 270.972,Z 347.643,A -85,B 0,C 180,E1 11241.782,E2 11241.782} C_VEL
LIN {X 0,Y 266.972,Z 342.496,A -85,B 0,C 180,E1 11239.209,E2 11239.209} C_VEL
LIN {X 0,Y 263.437,Z 337.732,A -85,B 0,C 180,E1 11236.616,E2 11236.616} C_VEL
LIN {X 0,Y 259.369,Z 332.938,A -85,B 0,C 180,E1 11233.428,E2 11233.428} C_VEL
LIN {X 0,Y 258.252,Z 331.288,A -85,B 0,C 180,E1 11232.426,E2 11232.426} C_VEL
LIN {X 0,Y 254.697,Z 327.404,A -85,B 0,C 180,E1 11229.192,E2 11229.192} C_VEL
LIN {X 0,Y 253.379,Z 325.235,A -85,B 0,C 180,E1 11227.742,E2 11227.742} C_VEL
LIN {X 0,Y 250.344,Z 322.42,A -85,B 0,C 180,E1 11224.45,E2 11224.45} C_VEL
LIN {X 0,Y 248.437,Z 319.049,A -85,B 0,C 180,E1 11221.801,E2 11221.801} C_VEL
LIN {X 0,Y 245.214,Z 316.617,A -85,B 0,C 180,E1 11217.128,E2 11217.128} C_VEL
LIN {X 0,Y 243.353,Z 312.808,A -85,B 0,C 180,E1 11212.715,E2 11212.715} C_VEL
LIN {X 0,Y 241.145,Z 311.648,A -85,B 0,C 180,E1 11206.169,E2 11206.169} C_VEL
LIN {X 0,Y 240.33,Z 311.013,A -85,B 0,C 180,E1 11199.838,E2 11199.838} C_VEL
LIN {X 0,Y 240.885,Z 311.478,A -85,B 0,C 180,E1 11193.503,E2 11193.503} C_VEL
LIN {X 0,Y 243.132,Z 312.586,A -85,B 0,C 180,E1 11186.304,E2 11186.304} C_VEL
LIN {X 0,Y 243.627,Z 313.728,A -85,B 0,C 180,E1 11184.914,E2 11184.914} C_VEL
LIN {X 0,Y 245.939,Z 317.428,A -85,B 0,C 180,E1 11180.104,E2 11180.104} C_VEL
LIN {X 0,Y 248.746,Z 319.51,A -85,B 0,C 180,E1 11176.13,E2 11176.13} C_VEL
LIN {X 0,Y 250.611,Z 322.955,A -85,B 0,C 180,E1 11173.376,E2 11173.376} C_VEL
LIN {X 0,Y 253.853,Z 325.872,A -85,B 0,C 180,E1 11169.919,E2 11169.919} C_VEL
LIN {X 0,Y 256.817,Z 330.141,A -85,B 0,C 180,E1 11166.912,E2 11166.912} C_VEL
LIN {X 0,Y 258.862,Z 332.106,A -85,B 0,C 180,E1 11165.094,E2 11165.094} C_VEL
LIN {X 0,Y 262.167,Z 336.537,A -85,B 0,C 180,E1 11162.337,E2 11162.337} C_VEL
LIN {X 0,Y 263.786,Z 338.345,A -85,B 0,C 180,E1 11161.083,E2 11161.083} C_VEL
LIN {X 0,Y 267.578,Z 343.014,A -85,B 0,C 180,E1 11158.391,E2 11158.391} C_VEL
LIN {X 0,Y 274.495,Z 352.241,A -85,B 0,C 180,E1 11153.914,E2 11153.914} C_VEL
LIN {X 0,Y 282.422,Z 364.088,A -85,B 0,C 180,E1 11149.389,E2 11149.389} C_VEL
LIN {X 0,Y 291.048,Z 377.224,A -85,B 0,C 180,E1 11145.118,E2 11145.118} C_VEL
LIN {X 0,Y 295.018,Z 383.579,A -85,B 0,C 180,E1 11143.31,E2 11143.31} C_VEL
LIN {X 0,Y 297.294,Z 388.517,A -85,B 0,C 180,E1 11142.243,E2 11142.243} C_VEL
LIN {X 0,Y 299.965,Z 399.034,A -85,B 0,C 180,E1 11140.724,E2 11140.724} C_VEL
LIN {X 0,Y 302.445,Z 407.67,A -85,B 0,C 180,E1 11139.437,E2 11139.437} C_VEL
LIN {X 0,Y 303.475,Z 409.903,A -85,B 0,C 180,E1 11139.003,E2 11139.003} C_VEL
LIN {X 0,Y 309.853,Z 421.567,A -85,B 0,C 180,E1 11136.56,E2 11136.56} C_VEL
LIN {X 0,Y 289.82,Z 591.297,A -85,B 0,C 180,E1 11131.963,E2 11131.963} C_VEL
LIN {X 0,Y 285.566,Z 615.165,A -85,B 0,C 180,E1 11131.045,E2 11131.045} C_VEL
LIN {X 0,Y 280.243,Z 637.719,A -85,B 0,C 180,E1 11129.9,E2 11129.9} C_VEL
LIN {X 0,Y 274.053,Z 659.874,A -85,B 0,C 180,E1 11128.414,E2 11128.414} C_VEL
LIN {X 0,Y 266.834,Z 682.219,A -85,B 0,C 180,E1 11126.479,E2 11126.479} C_VEL
LIN {X 0,Y 259.37,Z 702.687,A -85,B 0,C 180,E1 11124.235,E2 11124.235} C_VEL
LIN {X 0,Y 251.776,Z 721.703,A -85,B 0,C 180,E1 11121.637,E2 11121.637} C_VEL
LIN {X 0,Y 243.781,Z 740.318,A -85,B 0,C 180,E1 11118.458,E2 11118.458} C_VEL
LIN {X 0,Y 236.274,Z 756.748,A -85,B 0,C 180,E1 11114.963,E2 11114.963} C_VEL
LIN {X 0,Y 229.276,Z 771.773,A -85,B 0,C 180,E1 11111.02,E2 11111.02} C_VEL
LIN {X 0,Y 222.944,Z 785.414,A -85,B 0,C 180,E1 11106.6,E2 11106.6} C_VEL
LIN {X 0,Y 217.627,Z 797.399,A -85,B 0,C 180,E1 11101.789,E2 11101.789} C_VEL
LIN {X 0,Y 213.555,Z 807.446,A -85,B 0,C 180,E1 11096.706,E2 11096.706} C_VEL
LIN {X 0,Y 210.771,Z 815.724,A -85,B 0,C 180,E1 11091.421,E2 11091.421} C_VEL
LIN {X 0,Y 209.225,Z 822.231,A -85,B 0,C 180,E1 11086.089,E2 11086.089} C_VEL
LIN {X 0,Y 208.709,Z 826.697,A -85,B 0,C 180,E1 11081.045,E2 11081.045} C_VEL
LIN {X 0,Y 208.773,Z 829.735,A -85,B 0,C 180,E1 11076.045,E2 11076.045} C_VEL
LIN {X 0,Y 208.93,Z 831.084,A -85,B 0,C 180,E1 11071.643,E2 11071.643} C_VEL
LIN {X 0,Y 208.868,Z 831.319,A -85,B 0,C 180,E1 11067.528,E2 11067.528} C_VEL
LIN {X 0,Y 208.614,Z 830.408,A -85,B 0,C 180,E1 11062.822,E2 11062.822} C_VEL
LIN {X 0,Y 208.638,Z 827.724,A -85,B 0,C 180,E1 11057.262,E2 11057.262} C_VEL
LIN {X 0,Y 209.682,Z 823.299,A -85,B 0,C 180,E1 11051.366,E2 11051.366} C_VEL
LIN {X 0,Y 212.374,Z 816.746,A -85,B 0,C 180,E1 11045.225,E2 11045.225} C_VEL
LIN {X 0,Y 217.379,Z 807.787,A -85,B 0,C 180,E1 11038.823,E2 11038.823} C_VEL
LIN {X 0,Y 224.735,Z 796.933,A -85,B 0,C 180,E1 11032.763,E2 11032.763} C_VEL
LIN {X 0,Y 235.193,Z 783.365,A -85,B 0,C 180,E1 11026.805,E2 11026.805} C_VEL
LIN {X 0,Y 250.039,Z 766.127,A -85,B 0,C 180,E1 11020.904,E2 11020.904} C_VEL
LIN {X 0,Y 268.037,Z 747.377,A -85,B 0,C 180,E1 11015.953,E2 11015.953} C_VEL
LIN {X 0,Y 272.151,Z 743.301,A -85,B 0,C 180,E1 11015.01,E2 11015.01} C_VEL
LIN {X 0,Y 255.264,Z 756.648,A -85,B 0,C 180,E1 11010.353,E2 11010.353} C_VEL
LIN {X 0,Y 241.144,Z 768.125,A -85,B 0,C 180,E1 11005.022,E2 11005.022} C_VEL
LIN {X 0,Y 229.663,Z 777.632,A -85,B 0,C 180,E1 10999.061,E2 10999.061} C_VEL
LIN {X 0,Y 221.138,Z 784.827,A -85,B 0,C 180,E1 10992.803,E2 10992.803} C_VEL
LIN {X 0,Y 215.249,Z 789.848,A -85,B 0,C 180,E1 10986.404,E2 10986.404} C_VEL
LIN {X 0,Y 211.725,Z 792.778,A -85,B 0,C 180,E1 10980.274,E2 10980.274} C_VEL
LIN {X 0,Y 209.848,Z 794.095,A -85,B 0,C 180,E1 10974.261,E2 10974.261} C_VEL
LIN {X 0,Y 209.069,Z 794.002,A -85,B 0,C 180,E1 10968.647,E2 10968.647} C_VEL
LIN {X 0,Y 208.851,Z 792.633,A -85,B 0,C 180,E1 10963.597,E2 10963.597} C_VEL
LIN {X 0,Y 208.957,Z 790.134,A -85,B 0,C 180,E1 10958.385,E2 10958.385} C_VEL
LIN {X 0,Y 209.601,Z 786.105,A -85,B 0,C 180,E1 10953.057,E2 10953.057} C_VEL
LIN {X 0,Y 211.21,Z 780.193,A -85,B 0,C 180,E1 10947.344,E2 10947.344} C_VEL
LIN {X 0,Y 213.92,Z 772.797,A -85,B 0,C 180,E1 10941.911,E2 10941.911} C_VEL
LIN {X 0,Y 217.695,Z 763.893,A -85,B 0,C 180,E1 10936.822,E2 10936.822} C_VEL
LIN {X 0,Y 222.746,Z 752.988,A -85,B 0,C 180,E1 10931.836,E2 10931.836} C_VEL
LIN {X 0,Y 229.054,Z 739.896,A -85,B 0,C 180,E1 10927.044,E2 10927.044} C_VEL
LIN {X 0,Y 235.798,Z 725.891,A -85,B 0,C 180,E1 10922.912,E2 10922.912} C_VEL
LIN {X 0,Y 243.193,Z 710.075,A -85,B 0,C 180,E1 10919.131,E2 10919.131} C_VEL
LIN {X 0,Y 250.572,Z 693.281,A -85,B 0,C 180,E1 10915.884,E2 10915.884} C_VEL
LIN {X 0,Y 257.93,Z 675.342,A -85,B 0,C 180,E1 10913.051,E2 10913.051} C_VEL
LIN {X 0,Y 265.268,Z 655.702,A -85,B 0,C 180,E1 10910.522,E2 10910.522} C_VEL
LIN {X 0,Y 271.952,Z 635.747,A -85,B 0,C 180,E1 10908.434,E2 10908.434} C_VEL
LIN {X 0,Y 278.288,Z 614.022,A -85,B 0,C 180,E1 10906.616,E2 10906.616} C_VEL
LIN {X 0,Y 283.791,Z 591.527,A -85,B 0,C 180,E1 10905.14,E2 10905.14} C_VEL
LIN {X 0,Y 288.282,Z 568.949,A -85,B 0,C 180,E1 10903.997,E2 10903.997} C_VEL
LIN {X 0,Y 291.98,Z 544.699,A -85,B 0,C 180,E1 10903.099,E2 10903.099} C_VEL
LIN {X 0,Y 307.396,Z 411.232,A -85,B 0,C 180,E1 10899.503,E2 10899.503} C_VEL
LIN {X 0,Y 298.61,Z 397.449,A -85,B 0,C 180,E1 10896.206,E2 10896.206} C_VEL
LIN {X 0,Y 290.013,Z 384.593,A -85,B 0,C 180,E1 10892.62,E2 10892.62} C_VEL
LIN {X 0,Y 281.993,Z 373.243,A -85,B 0,C 180,E1 10888.886,E2 10888.886} C_VEL
LIN {X 0,Y 275.518,Z 364.32,A -85,B 0,C 180,E1 10885.48,E2 10885.48} C_VEL
LIN {X 0,Y 271.866,Z 359.535,A -85,B 0,C 180,E1 10883.456,E2 10883.456} C_VEL
LIN {X 0,Y 268.311,Z 354.738,A -85,B 0,C 180,E1 10881.214,E2 10881.214} C_VEL
LIN {X 0,Y 264.429,Z 349.704,A -85,B 0,C 180,E1 10878.663,E2 10878.663} C_VEL
LIN {X 0,Y 260.343,Z 344.397,A -85,B 0,C 180,E1 10875.66,E2 10875.66} C_VEL
LIN {X 0,Y 256.931,Z 340.025,A -85,B 0,C 180,E1 10872.8,E2 10872.8} C_VEL
LIN {X 0,Y 255.697,Z 338.561,A -85,B 0,C 180,E1 10871.773,E2 10871.773} C_VEL
LIN {X 0,Y 252.266,Z 334.372,A -85,B 0,C 180,E1 10868.434,E2 10868.434} C_VEL
LIN {X 0,Y 251.272,Z 332.853,A -85,B 0,C 180,E1 10867.383,E2 10867.383} C_VEL
LIN {X 0,Y 248.211,Z 329.824,A -85,B 0,C 180,E1 10863.926,E2 10863.926} C_VEL
LIN {X 0,Y 246.449,Z 326.735,A -85,B 0,C 180,E1 10861.4,E2 10861.4} C_VEL
LIN {X 0,Y 243.235,Z 324.113,A -85,B 0,C 180,E1 10856.552,E2 10856.552} C_VEL
LIN {X 0,Y 241.483,Z 320.41,A -85,B 0,C 180,E1 10852.212,E2 10852.212} C_VEL
LIN {X 0,Y 239.154,Z 319.269,A -85,B 0,C 180,E1 10844.95,E2 10844.95} C_VEL
LIN {X 0,Y 238.639,Z 318.843,A -85,B 0,C 180,E1 10839.189,E2 10839.189} C_VEL
LIN {X 0,Y 239.382,Z 319.436,A -85,B 0,C 180,E1 10832.598,E2 10832.598} C_VEL
LIN {X 0,Y 241.543,Z 320.582,A -85,B 0,C 180,E1 10826.022,E2 10826.022} C_VEL
LIN {X 0,Y 243.257,Z 324.295,A -85,B 0,C 180,E1 10821.707,E2 10821.707} C_VEL
LIN {X 0,Y 246.76,Z 327.18,A -85,B 0,C 180,E1 10816.474,E2 10816.474} C_VEL
LIN {X 0,Y 248.723,Z 330.676,A -85,B 0,C 180,E1 10813.598,E2 10813.598} C_VEL
LIN {X 0,Y 251.794,Z 333.482,A -85,B 0,C 180,E1 10810.29,E2 10810.29} C_VEL
LIN {X 0,Y 254.904,Z 337.887,A -85,B 0,C 180,E1 10807.097,E2 10807.097} C_VEL
LIN {X 0,Y 256.762,Z 339.788,A -85,B 0,C 180,E1 10805.415,E2 10805.415} C_VEL
LIN {X 0,Y 260.207,Z 344.252,A -85,B 0,C 180,E1 10802.546,E2 10802.546} C_VEL
LIN {X 0,Y 261.601,Z 345.971,A -85,B 0,C 180,E1 10801.421,E2 10801.421} C_VEL
LIN {X 0,Y 266.175,Z 351.766,A -85,B 0,C 180,E1 10798.131,E2 10798.131} C_VEL
LIN {X 0,Y 272.05,Z 359.75,A -85,B 0,C 180,E1 10794.302,E2 10794.302} C_VEL
LIN {X 0,Y 279.533,Z 371.013,A -85,B 0,C 180,E1 10789.955,E2 10789.955} C_VEL
LIN {X 0,Y 288.07,Z 384.22,A -85,B 0,C 180,E1 10785.628,E2 10785.628} C_VEL
LIN {X 0,Y 297.056,Z 398.936,A -85,B 0,C 180,E1 10781.604,E2 10781.604} C_VEL
LIN {X 0,Y 303.475,Z 409.903,A -85,B 0,C 180,E1 10779.003,E2 10779.003} C_VEL
LIN {X 0,Y 304.803,Z 414.023,A -85,B 0,C 180,E1 10778.379,E2 10778.379} C_VEL
LIN {X 0,Y 305.303,Z 420.087,A -85,B 0,C 180,E1 10777.878,E2 10777.878} C_VEL
LIN {X 0,Y 304.804,Z 427.865,A -85,B 0,C 180,E1 10777.55,E2 10777.55} C_VEL
LIN {X 0,Y 302.47,Z 444.345,A -85,B 0,C 180,E1 10777.198,E2 10777.198} C_VEL
LIN {X 0,Y 284.627,Z 590.507,A -85,B 0,C 180,E1 10773.184,E2 10773.184} C_VEL
LIN {X 0,Y 280.255,Z 614.393,A -85,B 0,C 180,E1 10772.259,E2 10772.259} C_VEL
LIN {X 0,Y 274.682,Z 637.364,A -85,B 0,C 180,E1 10771.091,E2 10771.091} C_VEL
LIN {X 0,Y 268.341,Z 659.407,A -85,B 0,C 180,E1 10769.603,E2 10769.603} C_VEL
LIN {X 0,Y 260.934,Z 681.7,A -85,B 0,C 180,E1 10767.658,E2 10767.658} C_VEL
LIN {X 0,Y 253.256,Z 702.146,A -85,B 0,C 180,E1 10765.397,E2 10765.397} C_VEL
LIN {X 0,Y 245.452,Z 721.1,A -85,B 0,C 180,E1 10762.781,E2 10762.781} C_VEL
LIN {X 0,Y 237.432,Z 739.182,A -85,B 0,C 180,E1 10759.655,E2 10759.655} C_VEL
LIN {X 0,Y 229.87,Z 755.207,A -85,B 0,C 180,E1 10756.219,E2 10756.219} C_VEL
LIN {X 0,Y 222.328,Z 770.828,A -85,B 0,C 180,E1 10752.07,E2 10752.07} C_VEL
LIN {X 0,Y 215.77,Z 784.397,A -85,B 0,C 180,E1 10747.586,E2 10747.586} C_VEL
LIN {X 0,Y 210.194,Z 796.409,A -85,B 0,C 180,E1 10742.648,E2 10742.648} C_VEL
LIN {X 0,Y 205.937,Z 806.377,A -85,B 0,C 180,E1 10737.464,E2 10737.464} C_VEL
LIN {X 0,Y 202.966,Z 814.738,A -85,B 0,C 180,E1 10731.984,E2 10731.984} C_VEL
LIN {X 0,Y 201.31,Z 821.309,A -85,B 0,C 180,E1 10726.442,E2 10726.442} C_VEL
LIN {X 0,Y 200.749,Z 825.851,A -85,B 0,C 180,E1 10721.12,E2 10721.12} C_VEL
LIN {X 0,Y 200.822,Z 828.872,A -85,B 0,C 180,E1 10715.999,E2 10715.999} C_VEL
LIN {X 0,Y 200.984,Z 830.229,A -85,B 0,C 180,E1 10711.422,E2 10711.422} C_VEL
LIN {X 0,Y 200.907,Z 830.473,A -85,B 0,C 180,E1 10707.43,E2 10707.43} C_VEL
LIN {X 0,Y 200.662,Z 829.777,A -85,B 0,C 180,E1 10703.129,E2 10703.129} C_VEL
LIN {X 0,Y 200.622,Z 827.588,A -85,B 0,C 180,E1 10697.623,E2 10697.623} C_VEL
LIN {X 0,Y 201.537,Z 823.644,A -85,B 0,C 180,E1 10691.784,E2 10691.784} C_VEL
LIN {X 0,Y 204.178,Z 817.686,A -85,B 0,C 180,E1 10685.4,E2 10685.4} C_VEL
LIN {X 0,Y 209.108,Z 809.526,A -85,B 0,C 180,E1 10678.863,E2 10678.863} C_VEL
LIN {X 0,Y 216.699,Z 799.135,A -85,B 0,C 180,E1 10672.476,E2 10672.476} C_VEL
LIN {X 0,Y 228.359,Z 785.308,A -85,B 0,C 180,E1 10665.877,E2 10665.877} C_VEL
LIN {X 0,Y 243.749,Z 769.048,A -85,B 0,C 180,E1 10659.905,E2 10659.905} C_VEL
LIN {X 0,Y 262.281,Z 751.537,A -85,B 0,C 180,E1 10654.951,E2 10654.951} C_VEL
LIN {X 0,Y 262.381,Z 751.425,A -85,B 0,C 180,E1 10654.865,E2 10654.865} C_VEL
LIN {X 0,Y 245.058,Z 763.796,A -85,B 0,C 180,E1 10649.855,E2 10649.855} C_VEL
LIN {X 0,Y 230.619,Z 774.35,A -85,B 0,C 180,E1 10644.053,E2 10644.053} C_VEL
LIN {X 0,Y 219.38,Z 782.684,A -85,B 0,C 180,E1 10637.715,E2 10637.715} C_VEL
LIN {X 0,Y 211.354,Z 788.674,A -85,B 0,C 180,E1 10631.187,E2 10631.187} C_VEL
LIN {X 0,Y 205.789,Z 792.776,A -85,B 0,C 180,E1 10624.183,E2 10624.183} C_VEL
LIN {X 0,Y 202.827,Z 794.705,A -85,B 0,C 180,E1 10617.744,E2 10617.744} C_VEL
LIN {X 0,Y 201.403,Z 795.057,A -85,B 0,C 180,E1 10611.439,E2 10611.439} C_VEL
LIN {X 0,Y 200.95,Z 794.138,A -85,B 0,C 180,E1 10605.893,E2 10605.893} C_VEL
LIN {X 0,Y 200.892,Z 791.941,A -85,B 0,C 180,E1 10600.525,E2 10600.525} C_VEL
LIN {X 0,Y 201.307,Z 788.521,A -85,B 0,C 180,E1 10595.032,E2 10595.032} C_VEL
LIN {X 0,Y 202.489,Z 783.47,A -85,B 0,C 180,E1 10589.435,E2 10589.435} C_VEL
LIN {X 0,Y 204.862,Z 776.543,A -85,B 0,C 180,E1 10583.643,E2 10583.643} C_VEL
LIN {X 0,Y 208.413,Z 768.154,A -85,B 0,C 180,E1 10578.182,E2 10578.182} C_VEL
LIN {X 0,Y 213.189,Z 758.012,A -85,B 0,C 180,E1 10572.983,E2 10572.983} C_VEL
LIN {X 0,Y 218.912,Z 746.416,A -85,B 0,C 180,E1 10568.232,E2 10568.232} C_VEL
LIN {X 0,Y 225.836,Z 732.598,A -85,B 0,C 180,E1 10563.668,E2 10563.668} C_VEL
LIN {X 0,Y 233.112,Z 717.789,A -85,B 0,C 180,E1 10559.718,E2 10559.718} C_VEL
LIN {X 0,Y 240.719,Z 701.624,A -85,B 0,C 180,E1 10556.22,E2 10556.22} C_VEL
LIN {X 0,Y 248.418,Z 683.97,A -85,B 0,C 180,E1 10553.13,E2 10553.13} C_VEL
LIN {X 0,Y 256.047,Z 664.949,A -85,B 0,C 180,E1 10550.427,E2 10550.427} C_VEL
LIN {X 0,Y 263.411,Z 644.581,A -85,B 0,C 180,E1 10548.087,E2 10548.087} C_VEL
LIN {X 0,Y 269.965,Z 624.06,A -85,B 0,C 180,E1 10546.184,E2 10546.184} C_VEL
LIN {X 0,Y 276.099,Z 601.609,A -85,B 0,C 180,E1 10544.527,E2 10544.527} C_VEL
LIN {X 0,Y 281.362,Z 578.042,A -85,B 0,C 180,E1 10543.188,E2 10543.188} C_VEL
LIN {X 0,Y 285.46,Z 554.691,A -85,B 0,C 180,E1 10542.204,E2 10542.204} C_VEL
LIN {X 0,Y 290.021,Z 518.878,A -85,B 0,C 180,E1 10541.148,E2 10541.148} C_VEL
LIN {X 0,Y 302.374,Z 415.301,A -85,B 0,C 180,E1 10538.368,E2 10538.368} C_VEL
LIN {X 0,Y 292.817,Z 400.25,A -85,B 0,C 180,E1 10534.614,E2 10534.614} C_VEL
LIN {X 0,Y 283.865,Z 386.949,A -85,B 0,C 180,E1 10530.663,E2 10530.663} C_VEL
LIN {X 0,Y 275.673,Z 375.446,A -85,B 0,C 180,E1 10526.571,E2 10526.571} C_VEL
LIN {X 0,Y 269.469,Z 366.974,A -85,B 0,C 180,E1 10523.076,E2 10523.076} C_VEL
LIN {X 0,Y 265.67,Z 361.898,A -85,B 0,C 180,E1 10520.689,E2 10520.689} C_VEL
LIN {X 0,Y 262.079,Z 357.087,A -85,B 0,C 180,E1 10518.225,E2 10518.225} C_VEL
LIN {X 0,Y 257.973,Z 351.767,A -85,B 0,C 180,E1 10515.181,E2 10515.181} C_VEL
LIN {X 0,Y 254.542,Z 347.299,A -85,B 0,C 180,E1 10512.279,E2 10512.279} C_VEL
LIN {X 0,Y 253.039,Z 345.669,A -85,B 0,C 180,E1 10510.977,E2 10510.977} C_VEL
LIN {X 0,Y 249.812,Z 341.375,A -85,B 0,C 180,E1 10507.717,E2 10507.717} C_VEL
LIN {X 0,Y 248.982,Z 340.346,A -85,B 0,C 180,E1 10506.827,E2 10506.827} C_VEL
LIN {X 0,Y 245.981,Z 337.129,A -85,B 0,C 180,E1 10503.326,E2 10503.326} C_VEL
LIN {X 0,Y 244.484,Z 334.43,A -85,B 0,C 180,E1 10501.058,E2 10501.058} C_VEL
LIN {X 0,Y 241.269,Z 331.601,A -85,B 0,C 180,E1 10495.971,E2 10495.971} C_VEL
LIN {X 0,Y 239.667,Z 328.191,A -85,B 0,C 180,E1 10491.875,E2 10491.875} C_VEL
LIN {X 0,Y 237.417,Z 327.049,A -85,B 0,C 180,E1 10484.687,E2 10484.687} C_VEL
LIN {X 0,Y 236.957,Z 326.668,A -85,B 0,C 180,E1 10478.95,E2 10478.95} C_VEL
LIN {X 0,Y 237.749,Z 327.288,A -85,B 0,C 180,E1 10472.278,E2 10472.278} C_VEL
LIN {X 0,Y 239.747,Z 328.38,A -85,B 0,C 180,E1 10466.232,E2 10466.232} C_VEL
LIN {X 0,Y 241.464,Z 332.061,A -85,B 0,C 180,E1 10461.877,E2 10461.877} C_VEL
LIN {X 0,Y 244.755,Z 334.787,A -85,B 0,C 180,E1 10456.857,E2 10456.857} C_VEL
LIN {X 0,Y 246.741,Z 338.28,A -85,B 0,C 180,E1 10453.948,E2 10453.948} C_VEL
LIN {X 0,Y 249.792,Z 341.182,A -85,B 0,C 180,E1 10450.607,E2 10450.607} C_VEL
LIN {X 0,Y 253.1,Z 345.758,A -85,B 0,C 180,E1 10447.157,E2 10447.157} C_VEL
LIN {X 0,Y 254.607,Z 347.348,A -85,B 0,C 180,E1 10445.801,E2 10445.801} C_VEL
LIN {X 0,Y 258.238,Z 352.006,A -85,B 0,C 180,E1 10442.706,E2 10442.706} C_VEL
LIN {X 0,Y 263.866,Z 359.335,A -85,B 0,C 180,E1 10438.477,E2 10438.477} C_VEL
LIN {X 0,Y 269.348,Z 366.869,A -85,B 0,C 180,E1 10434.833,E2 10434.833} C_VEL
LIN {X 0,Y 276.425,Z 377.635,A -85,B 0,C 180,E1 10430.63,E2 10430.63} C_VEL
LIN {X 0,Y 284.992,Z 391.047,A -85,B 0,C 180,E1 10426.195,E2 10426.195} C_VEL
LIN {X 0,Y 293.905,Z 405.887,A -85,B 0,C 180,E1 10422.117,E2 10422.117} C_VEL
LIN {X 0,Y 302.761,Z 421.419,A -85,B 0,C 180,E1 10418.493,E2 10418.493} C_VEL
LIN {X 0,Y 304.81,Z 425.431,A -85,B 0,C 180,E1 10417.687,E2 10417.687} C_VEL
LIN {X 0,Y 302.47,Z 444.345,A -85,B 0,C 180,E1 10417.198,E2 10417.198} C_VEL
LIN {X 0,Y 300.938,Z 451.956,A -85,B 0,C 180,E1 10417.156,E2 10417.156} C_VEL
LIN {X 0,Y 294.744,Z 472.153,A -85,B 0,C 180,E1 10417.601,E2 10417.601} C_VEL
LIN {X 0,Y 293.47,Z 478.683,A -85,B 0,C 180,E1 10417.545,E2 10417.545} C_VEL
LIN {X 0,Y 279.331,Z 590.518,A -85,B 0,C 180,E1 10414.403,E2 10414.403} C_VEL
LIN {X 0,Y 274.794,Z 614.535,A -85,B 0,C 180,E1 10413.466,E2 10413.466} C_VEL
LIN {X 0,Y 268.878,Z 638.127,A -85,B 0,C 180,E1 10412.25,E2 10412.25} C_VEL
LIN {X 0,Y 262.395,Z 659.868,A -85,B 0,C 180,E1 10410.757,E2 10410.757} C_VEL
LIN {X 0,Y 255.114,Z 681.122,A -85,B 0,C 180,E1 10408.883,E2 10408.883} C_VEL
LIN {X 0,Y 247.348,Z 701.236,A -85,B 0,C 180,E1 10406.647,E2 10406.647} C_VEL
LIN {X 0,Y 239.206,Z 720.427,A -85,B 0,C 180,E1 10403.975,E2 10403.975} C_VEL
LIN {X 0,Y 230.826,Z 738.714,A -85,B 0,C 180,E1 10400.768,E2 10400.768} C_VEL
LIN {X 0,Y 222.839,Z 755.051,A -85,B 0,C 180,E1 10397.185,E2 10397.185} C_VEL
LIN {X 0,Y 215.249,Z 770.173,A -85,B 0,C 180,E1 10393.061,E2 10393.061} C_VEL
LIN {X 0,Y 208.55,Z 783.493,A -85,B 0,C 180,E1 10388.551,E2 10388.551} C_VEL
LIN {X 0,Y 202.765,Z 795.403,A -85,B 0,C 180,E1 10383.52,E2 10383.52} C_VEL
LIN {X 0,Y 198.36,Z 805.217,A -85,B 0,C 180,E1 10378.279,E2 10378.279} C_VEL
LIN {X 0,Y 195.184,Z 813.682,A -85,B 0,C 180,E1 10372.591,E2 10372.591} C_VEL
LIN {X 0,Y 193.406,Z 820.325,A -85,B 0,C 180,E1 10366.825,E2 10366.825} C_VEL
LIN {X 0,Y 192.799,Z 824.863,A -85,B 0,C 180,E1 10361.362,E2 10361.362} C_VEL
LIN {X 0,Y 192.872,Z 827.988,A -85,B 0,C 180,E1 10355.948,E2 10355.948} C_VEL
LIN {X 0,Y 193.038,Z 829.361,A -85,B 0,C 180,E1 10351.184,E2 10351.184} C_VEL
LIN {X 0,Y 192.912,Z 829.593,A -85,B 0,C 180,E1 10346.729,E2 10346.729} C_VEL
LIN {X 0,Y 192.629,Z 828.752,A -85,B 0,C 180,E1 10341.941,E2 10341.941} C_VEL
LIN {X 0,Y 192.771,Z 826.245,A -85,B 0,C 180,E1 10335.888,E2 10335.888} C_VEL
LIN {X 0,Y 194.114,Z 822.175,A -85,B 0,C 180,E1 10329.809,E2 10329.809} C_VEL
LIN {X 0,Y 197.617,Z 815.744,A -85,B 0,C 180,E1 10322.909,E2 10322.909} C_VEL
LIN {X 0,Y 203.79,Z 807.195,A -85,B 0,C 180,E1 10316.018,E2 10316.018} C_VEL
LIN {X 0,Y 213.558,Z 795.76,A -85,B 0,C 180,E1 10309.042,E2 10309.042} C_VEL
LIN {X 0,Y 227.47,Z 781.466,A -85,B 0,C 180,E1 10302.397,E2 10302.397} C_VEL
LIN {X 0,Y 244.674,Z 765.647,A -85,B 0,C 180,E1 10296.776,E2 10296.776} C_VEL
LIN {X 0,Y 252.638,Z 758.87,A -85,B 0,C 180,E1 10294.746,E2 10294.746} C_VEL
LIN {X 0,Y 234.771,Z 770.355,A -85,B 0,C 180,E1 10289.328,E2 10289.328} C_VEL
LIN {X 0,Y 220.063,Z 779.97,A -85,B 0,C 180,E1 10283.004,E2 10283.004} C_VEL
LIN {X 0,Y 209.291,Z 787.044,A -85,B 0,C 180,E1 10276.375,E2 10276.375} C_VEL
LIN {X 0,Y 201.643,Z 791.975,A -85,B 0,C 180,E1 10269.421,E2 10269.421} C_VEL
LIN {X 0,Y 196.917,Z 794.828,A -85,B 0,C 180,E1 10262.623,E2 10262.623} C_VEL
LIN {X 0,Y 194.324,Z 795.996,A -85,B 0,C 180,E1 10255.873,E2 10255.873} C_VEL
LIN {X 0,Y 193.254,Z 795.749,A -85,B 0,C 180,E1 10249.873,E2 10249.873} C_VEL
LIN {X 0,Y 192.922,Z 794.267,A -85,B 0,C 180,E1 10244.37,E2 10244.37} C_VEL
LIN {X 0,Y 192.983,Z 791.673,A -85,B 0,C 180,E1 10238.74,E2 10238.74} C_VEL
LIN {X 0,Y 193.647,Z 787.568,A -85,B 0,C 180,E1 10232.981,E2 10232.981} C_VEL
LIN {X 0,Y 195.381,Z 781.553,A -85,B 0,C 180,E1 10226.805,E2 10226.805} C_VEL
LIN {X 0,Y 198.148,Z 774.533,A -85,B 0,C 180,E1 10221.272,E2 10221.272} C_VEL
LIN {X 0,Y 202.212,Z 765.6,A -85,B 0,C 180,E1 10215.805,E2 10215.805} C_VEL
LIN {X 0,Y 207.666,Z 754.689,A -85,B 0,C 180,E1 10210.479,E2 10210.479} C_VEL
LIN {X 0,Y 214.084,Z 742.323,A -85,B 0,C 180,E1 10205.652,E2 10205.652} C_VEL
LIN {X 0,Y 221.239,Z 728.535,A -85,B 0,C 180,E1 10201.316,E2 10201.316} C_VEL
LIN {X 0,Y 229.024,Z 712.936,A -85,B 0,C 180,E1 10197.39,E2 10197.39} C_VEL
LIN {X 0,Y 236.851,Z 696.367,A -85,B 0,C 180,E1 10194.01,E2 10194.01} C_VEL
LIN {X 0,Y 245.341,Z 677.01,A -85,B 0,C 180,E1 10190.831,E2 10190.831} C_VEL
LIN {X 0,Y 252.981,Z 657.811,A -85,B 0,C 180,E1 10188.293,E2 10188.293} C_VEL
LIN {X 0,Y 260.184,Z 637.589,A -85,B 0,C 180,E1 10186.127,E2 10186.127} C_VEL
LIN {X 0,Y 267.126,Z 615.087,A -85,B 0,C 180,E1 10184.218,E2 10184.218} C_VEL
LIN {X 0,Y 272.897,Z 592.759,A -85,B 0,C 180,E1 10182.738,E2 10182.738} C_VEL
LIN {X 0,Y 277.682,Z 570.071,A -85,B 0,C 180,E1 10181.579,E2 10181.579} C_VEL
LIN {X 0,Y 281.626,Z 545.804,A -85,B 0,C 180,E1 10180.67,E2 10180.67} C_VEL
LIN {X 0,Y 297.362,Z 419.382,A -85,B 0,C 180,E1 10177.23,E2 10177.23} C_VEL
LIN {X 0,Y 288.082,Z 404.79,A -85,B 0,C 180,E1 10173.434,E2 10173.434} C_VEL
LIN {X 0,Y 280.209,Z 392.944,A -85,B 0,C 180,E1 10169.798,E2 10169.798} C_VEL
LIN {X 0,Y 271.379,Z 380.222,A -85,B 0,C 180,E1 10165.194,E2 10165.194} C_VEL
LIN {X 0,Y 263.899,Z 370.008,A -85,B 0,C 180,E1 10160.681,E2 10160.681} C_VEL
LIN {X 0,Y 259.563,Z 364.28,A -85,B 0,C 180,E1 10157.658,E2 10157.658} C_VEL
LIN {X 0,Y 255.622,Z 359.134,A -85,B 0,C 180,E1 10154.694,E2 10154.694} C_VEL
LIN {X 0,Y 252.175,Z 354.573,A -85,B 0,C 180,E1 10151.749,E2 10151.749} C_VEL
LIN {X 0,Y 247.979,Z 349.447,A -85,B 0,C 180,E1 10147.662,E2 10147.662} C_VEL
LIN {X 0,Y 247.082,Z 348.074,A -85,B 0,C 180,E1 10146.639,E2 10146.639} C_VEL
LIN {X 0,Y 244.044,Z 344.849,A -85,B 0,C 180,E1 10143.085,E2 10143.085} C_VEL
LIN {X 0,Y 242.641,Z 342.184,A -85,B 0,C 180,E1 10140.87,E2 10140.87} C_VEL
LIN {X 0,Y 239.423,Z 339.292,A -85,B 0,C 180,E1 10135.686,E2 10135.686} C_VEL
LIN {X 0,Y 237.826,Z 335.968,A -85,B 0,C 180,E1 10131.525,E2 10131.525} C_VEL
LIN {X 0,Y 235.693,Z 334.848,A -85,B 0,C 180,E1 10124.55,E2 10124.55} C_VEL
LIN {X 0,Y 235.287,Z 334.493,A -85,B 0,C 180,E1 10118.569,E2 10118.569} C_VEL
LIN {X 0,Y 236.121,Z 335.15,A -85,B 0,C 180,E1 10111.954,E2 10111.954} C_VEL
LIN {X 0,Y 237.954,Z 336.179,A -85,B 0,C 180,E1 10106.445,E2 10106.445} C_VEL
LIN {X 0,Y 239.814,Z 339.993,A -85,B 0,C 180,E1 10101.778,E2 10101.778} C_VEL
LIN {X 0,Y 242.827,Z 342.574,A -85,B 0,C 180,E1 10097.118,E2 10097.118} C_VEL
LIN {X 0,Y 245.089,Z 346.289,A -85,B 0,C 180,E1 10093.86,E2 10093.86} C_VEL
LIN {X 0,Y 247.749,Z 348.851,A -85,B 0,C 180,E1 10090.931,E2 10090.931} C_VEL
LIN {X 0,Y 251.169,Z 353.513,A -85,B 0,C 180,E1 10087.315,E2 10087.315} C_VEL
LIN {X 0,Y 252.492,Z 354.992,A -85,B 0,C 180,E1 10086.135,E2 10086.135} C_VEL
LIN {X 0,Y 256.216,Z 359.711,A -85,B 0,C 180,E1 10082.905,E2 10082.905} C_VEL
LIN {X 0,Y 261.522,Z 366.851,A -85,B 0,C 180,E1 10078.847,E2 10078.847} C_VEL
LIN {X 0,Y 266.592,Z 373.85,A -85,B 0,C 180,E1 10075.426,E2 10075.426} C_VEL
LIN {X 0,Y 273.606,Z 384.672,A -85,B 0,C 180,E1 10071.169,E2 10071.169} C_VEL
LIN {X 0,Y 282.003,Z 398.017,A -85,B 0,C 180,E1 10066.725,E2 10066.725} C_VEL
LIN {X 0,Y 290.723,Z 412.809,A -85,B 0,C 180,E1 10062.639,E2 10062.639} C_VEL
LIN {X 0,Y 299.04,Z 427.646,A -85,B 0,C 180,E1 10059.138,E2 10059.138} C_VEL
LIN {X 0,Y 299.758,Z 429.315,A -85,B 0,C 180,E1 10058.833,E2 10058.833} C_VEL
LIN {X 0,Y 293.47,Z 478.683,A -85,B 0,C 180,E1 10057.545,E2 10057.545} C_VEL
LIN {X 0,Y 291.893,Z 486.284,A -85,B 0,C 180,E1 10057.497,E2 10057.497} C_VEL
LIN {X 0,Y 285.582,Z 506.446,A -85,B 0,C 180,E1 10057.953,E2 10057.953} C_VEL
LIN {X 0,Y 284.314,Z 512.977,A -85,B 0,C 180,E1 10057.898,E2 10057.898} C_VEL
LIN {X 0,Y 274.199,Z 590.33,A -85,B 0,C 180,E1 10055.676,E2 10055.676} C_VEL
LIN {X 0,Y 269.644,Z 613.809,A -85,B 0,C 180,E1 10054.756,E2 10054.756} C_VEL
LIN {X 0,Y 263.764,Z 636.742,A -85,B 0,C 180,E1 10053.583,E2 10053.583} C_VEL
LIN {X 0,Y 257.235,Z 658.206,A -85,B 0,C 180,E1 10052.126,E2 10052.126} C_VEL
LIN {X 0,Y 249.368,Z 680.63,A -85,B 0,C 180,E1 10050.152,E2 10050.152} C_VEL
LIN {X 0,Y 241.384,Z 700.717,A -85,B 0,C 180,E1 10047.903,E2 10047.903} C_VEL
LIN {X 0,Y 232.92,Z 720.043,A -85,B 0,C 180,E1 10045.182,E2 10045.182} C_VEL
LIN {X 0,Y 224.32,Z 738.203,A -85,B 0,C 180,E1 10041.951,E2 10041.951} C_VEL
LIN {X 0,Y 216.13,Z 754.383,A -85,B 0,C 180,E1 10038.337,E2 10038.337} C_VEL
LIN {X 0,Y 208.238,Z 769.519,A -85,B 0,C 180,E1 10034.12,E2 10034.12} C_VEL
LIN {X 0,Y 201.257,Z 782.842,A -85,B 0,C 180,E1 10029.483,E2 10029.483} C_VEL
LIN {X 0,Y 195.214,Z 794.754,A -85,B 0,C 180,E1 10024.287,E2 10024.287} C_VEL
LIN {X 0,Y 190.578,Z 804.626,A -85,B 0,C 180,E1 10018.812,E2 10018.812} C_VEL
LIN {X 0,Y 187.287,Z 813.005,A -85,B 0,C 180,E1 10012.933,E2 10012.933} C_VEL
LIN {X 0,Y 185.443,Z 819.621,A -85,B 0,C 180,E1 10006.924,E2 10006.924} C_VEL
LIN {X 0,Y 184.837,Z 824.12,A -85,B 0,C 180,E1 10001.226,E2 10001.226} C_VEL
LIN {X 0,Y 184.932,Z 827.095,A -85,B 0,C 180,E1 9995.807,E2 9995.807} C_VEL
LIN {X 0,Y 185.092,Z 828.484,A -85,B 0,C 180,E1 9990.925,E2 9990.925} C_VEL
LIN {X 0,Y 184.929,Z 828.716,A -85,B 0,C 180,E1 9986.277,E2 9986.277} C_VEL
LIN {X 0,Y 184.641,Z 827.967,A -85,B 0,C 180,E1 9981.59,E2 9981.59} C_VEL
LIN {X 0,Y 184.809,Z 825.763,A -85,B 0,C 180,E1 9975.576,E2 9975.576} C_VEL
LIN {X 0,Y 186.492,Z 821.434,A -85,B 0,C 180,E1 9968.616,E2 9968.616} C_VEL
LIN {X 0,Y 190.762,Z 814.764,A -85,B 0,C 180,E1 9961.088,E2 9961.088} C_VEL
LIN {X 0,Y 197.793,Z 806.324,A -85,B 0,C 180,E1 9953.984,E2 9953.984} C_VEL
LIN {X 0,Y 209.243,Z 794.529,A -85,B 0,C 180,E1 9946.583,E2 9946.583} C_VEL
LIN {X 0,Y 224.538,Z 780.664,A -85,B 0,C 180,E1 9940.009,E2 9940.009} C_VEL
LIN {X 0,Y 242.803,Z 765.765,A -85,B 0,C 180,E1 9934.633,E2 9934.633} C_VEL
LIN {X 0,Y 224.979,Z 776.012,A -85,B 0,C 180,E1 9928.978,E2 9928.978} C_VEL
LIN {X 0,Y 210.365,Z 784.464,A -85,B 0,C 180,E1 9922.352,E2 9922.352} C_VEL
LIN {X 0,Y 199.794,Z 790.505,A -85,B 0,C 180,E1 9915.385,E2 9915.385} C_VEL
LIN {X 0,Y 192.685,Z 794.376,A -85,B 0,C 180,E1 9908.358,E2 9908.358} C_VEL
LIN {X 0,Y 188.246,Z 796.491,A -85,B 0,C 180,E1 9901.221,E2 9901.221} C_VEL
LIN {X 0,Y 186.093,Z 797.041,A -85,B 0,C 180,E1 9894.764,E2 9894.764} C_VEL
LIN {X 0,Y 185.177,Z 796.237,A -85,B 0,C 180,E1 9888.796,E2 9888.796} C_VEL
LIN {X 0,Y 184.931,Z 794.447,A -85,B 0,C 180,E1 9883.029,E2 9883.029} C_VEL
LIN {X 0,Y 185.112,Z 791.27,A -85,B 0,C 180,E1 9877.119,E2 9877.119} C_VEL
LIN {X 0,Y 186.053,Z 786.723,A -85,B 0,C 180,E1 9871.081,E2 9871.081} C_VEL
LIN {X 0,Y 188.115,Z 780.491,A -85,B 0,C 180,E1 9864.974,E2 9864.974} C_VEL
LIN {X 0,Y 191.355,Z 772.861,A -85,B 0,C 180,E1 9859.228,E2 9859.228} C_VEL
LIN {X 0,Y 196.101,Z 763.256,A -85,B 0,C 180,E1 9853.501,E2 9853.501} C_VEL
LIN {X 0,Y 202.12,Z 751.913,A -85,B 0,C 180,E1 9848.144,E2 9848.144} C_VEL
LIN {X 0,Y 209.192,Z 738.752,A -85,B 0,C 180,E1 9843.243,E2 9843.243} C_VEL
LIN {X 0,Y 216.799,Z 724.41,A -85,B 0,C 180,E1 9838.966,E2 9838.966} C_VEL
LIN {X 0,Y 225.396,Z 707.504,A -85,B 0,C 180,E1 9834.927,E2 9834.927} C_VEL
LIN {X 0,Y 233.743,Z 690.023,A -85,B 0,C 180,E1 9831.587,E2 9831.587} C_VEL
LIN {X 0,Y 241.791,Z 671.718,A -85,B 0,C 180,E1 9828.758,E2 9828.758} C_VEL
LIN {X 0,Y 249.886,Z 651.158,A -85,B 0,C 180,E1 9826.214,E2 9826.214} C_VEL
LIN {X 0,Y 257.189,Z 630.113,A -85,B 0,C 180,E1 9824.141,E2 9824.141} C_VEL
LIN {X 0,Y 263.761,Z 608.13,A -85,B 0,C 180,E1 9822.421,E2 9822.421} C_VEL
LIN {X 0,Y 269.534,Z 584.916,A -85,B 0,C 180,E1 9821.002,E2 9821.002} C_VEL
LIN {X 0,Y 274.192,Z 561.516,A -85,B 0,C 180,E1 9819.925,E2 9819.925} C_VEL
LIN {X 0,Y 277.816,Z 537.31,A -85,B 0,C 180,E1 9819.126,E2 9819.126} C_VEL
LIN {X 0,Y 292.36,Z 423.462,A -85,B 0,C 180,E1 9816.038,E2 9816.038} C_VEL
LIN {X 0,Y 283.346,Z 409.122,A -85,B 0,C 180,E1 9812.176,E2 9812.176} C_VEL
LIN {X 0,Y 274.667,Z 396.112,A -85,B 0,C 180,E1 9807.968,E2 9807.968} C_VEL
LIN {X 0,Y 267.522,Z 385.923,A -85,B 0,C 180,E1 9804.049,E2 9804.049} C_VEL
LIN {X 0,Y 261.467,Z 377.381,A -85,B 0,C 180,E1 9800.26,E2 9800.26} C_VEL
LIN {X 0,Y 256.933,Z 371.414,A -85,B 0,C 180,E1 9797.072,E2 9797.072} C_VEL
LIN {X 0,Y 253.291,Z 366.497,A -85,B 0,C 180,E1 9794.197,E2 9794.197} C_VEL
LIN {X 0,Y 249.123,Z 361.083,A -85,B 0,C 180,E1 9790.544,E2 9790.544} C_VEL
LIN {X 0,Y 245.637,Z 356.584,A -85,B 0,C 180,E1 9787.001,E2 9787.001} C_VEL
LIN {X 0,Y 244.538,Z 355.312,A -85,B 0,C 180,E1 9785.743,E2 9785.743} C_VEL
LIN {X 0,Y 241.355,Z 351.222,A -85,B 0,C 180,E1 9781.687,E2 9781.687} C_VEL
LIN {X 0,Y 240.583,Z 349.809,A -85,B 0,C 180,E1 9780.362,E2 9780.362} C_VEL
LIN {X 0,Y 237.421,Z 346.823,A -85,B 0,C 180,E1 9775.198,E2 9775.198} C_VEL
LIN {X 0,Y 236.102,Z 343.78,A -85,B 0,C 180,E1 9771.503,E2 9771.503} C_VEL
LIN {X 0,Y 233.949,Z 342.648,A -85,B 0,C 180,E1 9764.465,E2 9764.465} C_VEL
LIN {X 0,Y 233.57,Z 342.308,A -85,B 0,C 180,E1 9758.363,E2 9758.363} C_VEL
LIN {X 0,Y 234.497,Z 343.033,A -85,B 0,C 180,E1 9751.492,E2 9751.492} C_VEL
LIN {X 0,Y 236.136,Z 343.966,A -85,B 0,C 180,E1 9746.664,E2 9746.664} C_VEL
LIN {X 0,Y 238.043,Z 347.816,A -85,B 0,C 180,E1 9741.841,E2 9741.841} C_VEL
LIN {X 0,Y 240.884,Z 350.34,A -85,B 0,C 180,E1 9737.385,E2 9737.385} C_VEL
LIN {X 0,Y 243.418,Z 354.279,A -85,B 0,C 180,E1 9733.779,E2 9733.779} C_VEL
LIN {X 0,Y 245.669,Z 356.517,A -85,B 0,C 180,E1 9731.246,E2 9731.246} C_VEL
LIN {X 0,Y 249.213,Z 361.24,A -85,B 0,C 180,E1 9727.501,E2 9727.501} C_VEL
LIN {X 0,Y 250.768,Z 363.311,A -85,B 0,C 180,E1 9726.062,E2 9726.062} C_VEL
LIN {X 0,Y 254.732,Z 368.4,A -85,B 0,C 180,E1 9722.64,E2 9722.64} C_VEL
LIN {X 0,Y 259.043,Z 374.135,A -85,B 0,C 180,E1 9719.334,E2 9719.334} C_VEL
LIN {X 0,Y 264.008,Z 381.098,A -85,B 0,C 180,E1 9715.925,E2 9715.925} C_VEL
LIN {X 0,Y 271.043,Z 392.113,A -85,B 0,C 180,E1 9711.565,E2 9711.565} C_VEL
LIN {X 0,Y 279.086,Z 405.122,A -85,B 0,C 180,E1 9707.216,E2 9707.216} C_VEL
LIN {X 0,Y 287.519,Z 419.706,A -85,B 0,C 180,E1 9703.169,E2 9703.169} C_VEL
LIN {X 0,Y 294.839,Z 432.852,A -85,B 0,C 180,E1 9700.024,E2 9700.024} C_VEL
LIN {X 0,Y 284.314,Z 512.977,A -85,B 0,C 180,E1 9697.898,E2 9697.898} C_VEL
LIN {X 0,Y 282.751,Z 520.58,A -85,B 0,C 180,E1 9697.851,E2 9697.851} C_VEL
LIN {X 0,Y 276.345,Z 540.719,A -85,B 0,C 180,E1 9698.315,E2 9698.315} C_VEL
LIN {X 0,Y 275.033,Z 547.244,A -85,B 0,C 180,E1 9698.255,E2 9698.255} C_VEL
LIN {X 0,Y 268.867,Z 591.404,A -85,B 0,C 180,E1 9696.93,E2 9696.93} C_VEL
LIN {X 0,Y 264.251,Z 614.229,A -85,B 0,C 180,E1 9696.025,E2 9696.025} C_VEL
LIN {X 0,Y 258.001,Z 637.737,A -85,B 0,C 180,E1 9694.804,E2 9694.804} C_VEL
LIN {X 0,Y 251.213,Z 659.216,A -85,B 0,C 180,E1 9693.315,E2 9693.315} C_VEL
LIN {X 0,Y 243.595,Z 680.222,A -85,B 0,C 180,E1 9691.442,E2 9691.442} C_VEL
LIN {X 0,Y 235.262,Z 700.566,A -85,B 0,C 180,E1 9689.142,E2 9689.142} C_VEL
LIN {X 0,Y 226.731,Z 719.46,A -85,B 0,C 180,E1 9686.451,E2 9686.451} C_VEL
LIN {X 0,Y 217.895,Z 737.528,A -85,B 0,C 180,E1 9683.195,E2 9683.195} C_VEL
LIN {X 0,Y 209.25,Z 754.034,A -85,B 0,C 180,E1 9679.437,E2 9679.437} C_VEL
LIN {X 0,Y 201.305,Z 768.701,A -85,B 0,C 180,E1 9675.252,E2 9675.252} C_VEL
LIN {X 0,Y 194.024,Z 782.057,A -85,B 0,C 180,E1 9670.485,E2 9670.485} C_VEL
LIN {X 0,Y 187.705,Z 793.984,A -85,B 0,C 180,E1 9665.116,E2 9665.116} C_VEL
LIN {X 0,Y 182.878,Z 803.804,A -85,B 0,C 180,E1 9659.472,E2 9659.472} C_VEL
LIN {X 0,Y 179.291,Z 812.562,A -85,B 0,C 180,E1 9653.043,E2 9653.043} C_VEL
LIN {X 0,Y 177.486,Z 818.865,A -85,B 0,C 180,E1 9647.03,E2 9647.03} C_VEL
LIN {X 0,Y 176.879,Z 823.349,A -85,B 0,C 180,E1 9641.077,E2 9641.077} C_VEL
LIN {X 0,Y 176.998,Z 826.258,A -85,B 0,C 180,E1 9635.507,E2 9635.507} C_VEL
LIN {X 0,Y 177.151,Z 827.629,A -85,B 0,C 180,E1 9630.32,E2 9630.32} C_VEL
LIN {X 0,Y 176.923,Z 827.813,A -85,B 0,C 180,E1 9625.459,E2 9625.459} C_VEL
LIN {X 0,Y 176.63,Z 826.899,A -85,B 0,C 180,E1 9620.071,E2 9620.071} C_VEL
LIN {X 0,Y 177.151,Z 824.305,A -85,B 0,C 180,E1 9613.268,E2 9613.268} C_VEL
LIN {X 0,Y 179.55,Z 819.786,A -85,B 0,C 180,E1 9606.011,E2 9606.011} C_VEL
LIN {X 0,Y 185.086,Z 812.732,A -85,B 0,C 180,E1 9598.031,E2 9598.031} C_VEL
LIN {X 0,Y 193.786,Z 803.871,A -85,B 0,C 180,E1 9590.604,E2 9590.604} C_VEL
LIN {X 0,Y 207.711,Z 791.597,A -85,B 0,C 180,E1 9582.969,E2 9582.969} C_VEL
LIN {X 0,Y 226.706,Z 776.704,A -85,B 0,C 180,E1 9576.183,E2 9576.183} C_VEL
LIN {X 0,Y 232.731,Z 772.211,A -85,B 0,C 180,E1 9574.476,E2 9574.476} C_VEL
LIN {X 0,Y 214.562,Z 781.492,A -85,B 0,C 180,E1 9568.384,E2 9568.384} C_VEL
LIN {X 0,Y 200.185,Z 788.767,A -85,B 0,C 180,E1 9561.387,E2 9561.387} C_VEL
LIN {X 0,Y 190.278,Z 793.586,A -85,B 0,C 180,E1 9554.302,E2 9554.302} C_VEL
LIN {X 0,Y 183.301,Z 796.692,A -85,B 0,C 180,E1 9546.582,E2 9546.582} C_VEL
LIN {X 0,Y 179.26,Z 797.937,A -85,B 0,C 180,E1 9538.726,E2 9538.726} C_VEL
LIN {X 0,Y 177.584,Z 797.625,A -85,B 0,C 180,E1 9531.913,E2 9531.913} C_VEL
LIN {X 0,Y 177.019,Z 795.991,A -85,B 0,C 180,E1 9525.615,E2 9525.615} C_VEL
LIN {X 0,Y 176.994,Z 793.35,A -85,B 0,C 180,E1 9519.503,E2 9519.503} C_VEL
LIN {X 0,Y 177.618,Z 789.208,A -85,B 0,C 180,E1 9513.24,E2 9513.24} C_VEL
LIN {X 0,Y 179.428,Z 783.166,A -85,B 0,C 180,E1 9506.524,E2 9506.524} C_VEL
LIN {X 0,Y 182.392,Z 776.109,A -85,B 0,C 180,E1 9500.52,E2 9500.52} C_VEL
LIN {X 0,Y 186.898,Z 766.935,A -85,B 0,C 180,E1 9494.496,E2 9494.496} C_VEL
LIN {X 0,Y 192.729,Z 756.133,A -85,B 0,C 180,E1 9488.886,E2 9488.886} C_VEL
LIN {X 0,Y 199.895,Z 743.321,A -85,B 0,C 180,E1 9483.62,E2 9483.62} C_VEL
LIN {X 0,Y 207.551,Z 729.586,A -85,B 0,C 180,E1 9479.117,E2 9479.117} C_VEL
LIN {X 0,Y 216.263,Z 713.277,A -85,B 0,C 180,E1 9474.883,E2 9474.883} C_VEL
LIN {X 0,Y 224.68,Z 696.48,A -85,B 0,C 180,E1 9471.405,E2 9471.405} C_VEL
LIN {X 0,Y 233.251,Z 678.016,A -85,B 0,C 180,E1 9468.333,E2 9468.333} C_VEL
LIN {X 0,Y 241.504,Z 658.383,A -85,B 0,C 180,E1 9465.708,E2 9465.708} C_VEL
LIN {X 0,Y 249.152,Z 637.97,A -85,B 0,C 180,E1 9463.516,E2 9463.516} C_VEL
LIN {X 0,Y 256.457,Z 615.496,A -85,B 0,C 180,E1 9461.607,E2 9461.607} C_VEL
LIN {X 0,Y 262.733,Z 592.364,A -85,B 0,C 180,E1 9460.084,E2 9460.084} C_VEL
LIN {X 0,Y 267.753,Z 569.448,A -85,B 0,C 180,E1 9458.931,E2 9458.931} C_VEL
LIN {X 0,Y 271.75,Z 545.855,A -85,B 0,C 180,E1 9458.06,E2 9458.06} C_VEL
LIN {X 0,Y 287.473,Z 427.515,A -85,B 0,C 180,E1 9454.79,E2 9454.79} C_VEL
LIN {X 0,Y 277.837,Z 412.202,A -85,B 0,C 180,E1 9450.466,E2 9450.466} C_VEL
LIN {X 0,Y 268.974,Z 398.93,A -85,B 0,C 180,E1 9445.899,E2 9445.899} C_VEL
LIN {X 0,Y 261.667,Z 388.546,A -85,B 0,C 180,E1 9441.554,E2 9441.554} C_VEL
LIN {X 0,Y 255.32,Z 379.622,A -85,B 0,C 180,E1 9437.17,E2 9437.17} C_VEL
LIN {X 0,Y 250.774,Z 373.671,A -85,B 0,C 180,E1 9433.558,E2 9433.558} C_VEL
LIN {X 0,Y 246.959,Z 368.584,A -85,B 0,C 180,E1 9430.12,E2 9430.12} C_VEL
LIN {X 0,Y 243.275,Z 363.6,A -85,B 0,C 180,E1 9426.251,E2 9426.251} C_VEL
LIN {X 0,Y 239.784,Z 359.617,A -85,B 0,C 180,E1 9421.986,E2 9421.986} C_VEL
LIN {X 0,Y 238.652,Z 357.518,A -85,B 0,C 180,E1 9420.098,E2 9420.098} C_VEL
LIN {X 0,Y 235.528,Z 354.499,A -85,B 0,C 180,E1 9414.903,E2 9414.903} C_VEL
